// TIA Portal V20 export
FUNCTION_BLOCK "CallUnit"   // FB130, LAD
TITLE = CallUnit
// This block calls all functionality inside the unit.
// stored: IsIECCheckEnabled true, MemoryReserve 100, Namespace Unit1, SetENOAutomatically true
   VAR_INPUT
      safetyReleased : Bool;   // Status from safety program
   END_VAR
   VAR_OUTPUT
      acknowledgeSafety { ExternalWritable := 'False'} : Bool;   // Acknowledge command to the safety program
   END_VAR
   VAR_IN_OUT
      globalStatus : "LAF_typeGeneralStatus";   // Global status
      unitInterface : "LAF_typeUnitInterface";   // Global unit interface
   END_VAR
   VAR
      instManageAlarms { ExternalWritable := 'False'} : "LAF_ManageAlarms";
      instStatusCollector { ExternalWritable := 'False'} : "LUC_StatusCollector";
      instInterfaceManager { ExternalWritable := 'False'} : "LUC_InterfaceManager";
      instUnitModeStateManager { ExternalWritable := 'False'} : "LPMLV2022_UnitModeStateManager";
      instRemoteInterfaceOpcUa { ExternalWritable := 'False'} : "LUC_RemoteCtrl_OpcUa";
      instSignalStack { ExternalWritable := 'False'} : "LUC_SignalStack";
      instUnitModeStateTimes { ExternalWritable := 'False'} : "LPMLV2022_UnitModeStateTimes";
      instUnitModeChangeAllowed { ExternalWritable := 'False'} : "LPMLV2022_UnitModeChangeAllowed";
      instPFEEvents { ExternalWritable := 'False'} : "Unit1.EventsPFE";
      instEQP_Interface_BA030 { ExternalWritable := 'False'} : "LER_EQP_Interface";
      instEQP_Interface_BA040 { ExternalWritable := 'False'} : "LER_EQP_Interface";
      instEQP_Interface_BA100 { S7_SetPoint := 'True'} : "LER_EQP_m_Interface";
      instEQP_Interface_CoveyorA { ExternalWritable := 'False'} : "LER_EQP_Communication";
      instSinaInfeed { ExternalWritable := 'False'} : SinaInfeed;
      statRemoteInterface { ExternalWritable := 'False'} : "LUC_typeCommands";
      statLocalInterface { ExternalWritable := 'False'} : "LUC_typeCommands";
      statEmEnableCheck { ExternalWritable := 'False'} : Array[0..2] of Bool;
      statEmHomeScCheck { ExternalWritable := 'False'} : Array[0..9] of Bool;
      statRunOutStatusCheck { ExternalWritable := 'False'} : Array[0..9] of Bool;
      statEOCStatusCheck { ExternalWritable := 'False'} : Array[0..19] of Bool;
      statPartData { ExternalWritable := 'False'} : Struct
         BA030 : "LER_typePartData";
         BA040 : "LER_typePartData";
      END_STRUCT;
      statDataDelete { ExternalWritable := 'False'} : "LER_typePartData";
      statTonTime { ExternalWritable := 'False'} : Array[0..99] of TON_TIME;
      statTofTime { ExternalWritable := 'False'} : Array[0..9] of TOF_TIME;
      statFlipFlop { ExternalWritable := 'False'} : Array[0..99] of Bool;
      statPulse { ExternalWritable := 'False'} : Array[0..9999] of Bool;
      statNoModeCmd { ExternalWritable := 'False'} : Bool;
      statEnableManualCmds { ExternalWritable := 'False'} : Bool;
      InstLER_FFU_LIU117 { S7_SetPoint := 'True'} : "LER_FFU_LIU117";
      ClearData { S7_SetPoint := 'True'} : "LER_typePartData";
      Data_TrCondition { S7_SetPoint := 'True'} : Array[0..20] of Bool;
      NoData_Alarm : Array[0..20] of Bool;
      statAllEmLinked : Bool;
      citi_Ptrig : Array[0..20] of Bool;
      citiTon : Array[0..20] of TON_TIME;
      citi : Time;
      citiTest : Array[0..20] of Bool;
      instMQTTClient { S7_SetPoint := 'True'} : "LMQTT_Client";
      instPFEUnit { S7_SetPoint := 'True'} : "Unit1.EventsPFE_Unit";
   END_VAR
   VAR_TEMP
      tempUnitFeedback : "LUC_typeEmFeedback";   // Collected commands in the unit, e.g. direct command or commands derived from alarms
      tempProcessCommands : "LUC_typeStateCommands";   // Requested unit state changes by the process
      tempUnitMode : DInt;   // Requested unit mode
      tempUnitModeChangeRequest : Bool;   // Request unit mode
      tempCntrlCmd : DInt;   // Request control command
      tempCmdChangeRequest : Bool;   // Enable change into requested state
      tempSc : Bool;   // State change from FALSE to TRUE (rising edge) triggers state complete signal
      tempEM_Linked_Status_1 : Bool;
      tempEM_Linked_Status_2 : Bool;
      tempDeleteData : Bool;
      tempGather8bits : Array[0..7] of Bool;
   END_VAR
   VAR CONSTANT
      delayTime : Time := T#2s;
      TRUE : Bool := TRUE;
      FALSE : Bool := FALSE;
   END_VAR
   VAR_TEMP   // added for the SCL form of the ladder/FBD networks
      _w1 : Bool;
      _w2 : Bool;
      _w3 : Bool;
      _w4 : Bool;
      _w5 : Bool;
      _w6 : Bool;
      _w7 : Bool;
      _w8 : Bool;
   END_VAR
BEGIN

REGION Network 1: BLOCK INFO HEADER
   // (company) / (C) Copyright (year)
   // ---------------------------------------------------------------------------------
   // Title:                             (Title of this block)
   // Comment/Function: (that is implemented in the block)
   // Library/Family:           (that the source is dedicated to)
   // Author:                        (department / person in charge / contact)
   // Target System:          (test system with FW version)
   // Engineering:              TIA Portal (SW version)
   // Restrictions:               (OB types, etc.)
   // Requirements:           (hardware, technological package, etc.)
   // ---------------------------------------------------------------------------------
   // Change log table:
   // Version          | Date             | Signature      | Expert in charge  | Changes applied ------------------------|----------------------|-------------------------|--------------------------------|-----------------------
   // 001.000.000 | yyyy-mm-dd | 0x00000000 | (name of expert) | First released version
END_REGION

REGION Network 2: DESCRIPTION
   // This is a template block provided by the Automation Framework. It can be used to create an own project.
   // The Block Info Header is prepared to put in your own data.
   // Description of the block could be added here and the docu created by Code2Docu.
END_REGION

REGION Network 3: Simulation
   // If simulation is active on a global level, inherit this status and set simulation active in this unit also. Information is written to DB ControlNodes, from where it is distributed to the equipmemt modules.
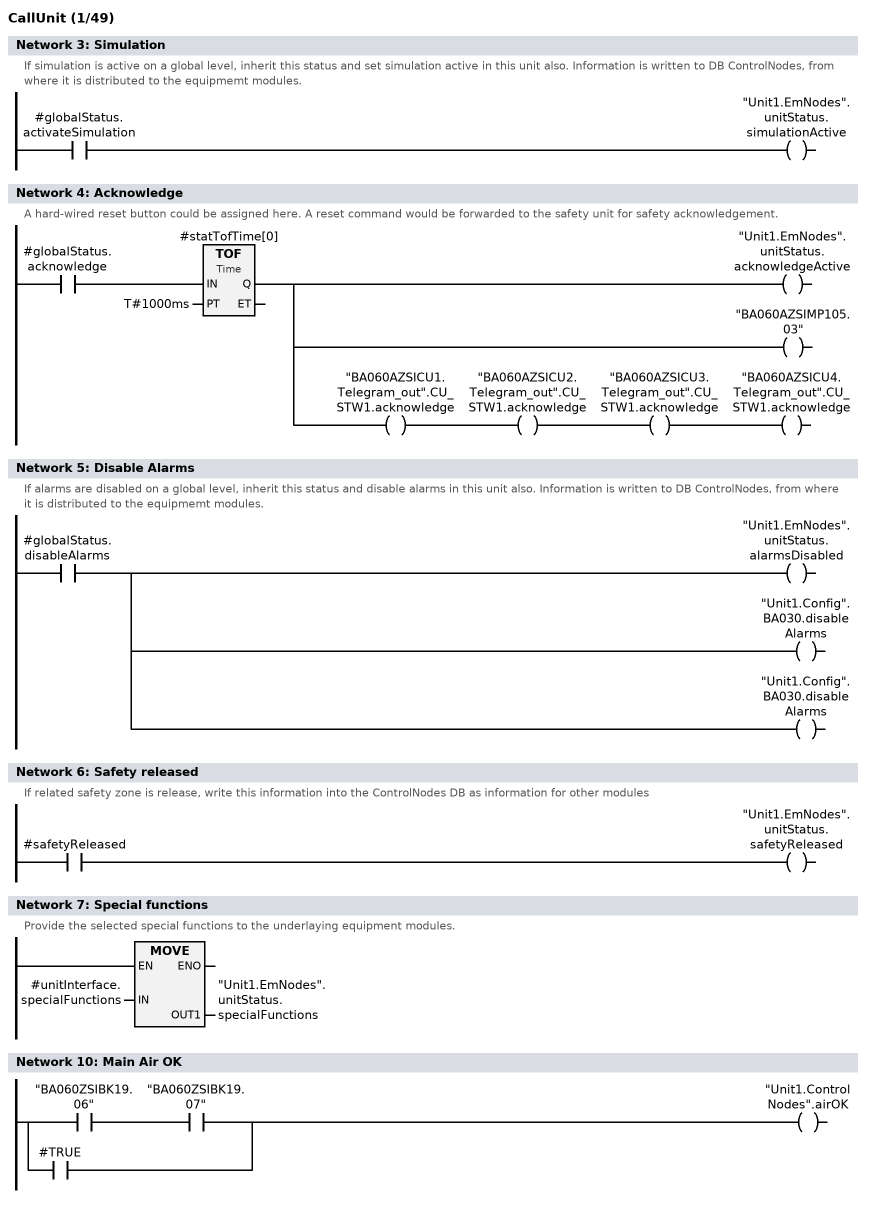
   RUNG wire#powerrail
      Contact( #globalStatus.activateSimulation )
      Coil( "Unit1.EmNodes".unitStatus.simulationActive )
   END_RUNG
   // the same network as SCL:
   "Unit1.EmNodes".unitStatus.simulationActive := #globalStatus.activateSimulation;
END_REGION

REGION Network 4: Acknowledge
   // A hard-wired reset button could be assigned here. A reset command would be forwarded to the safety unit for safety acknowledgement.
   RUNG wire#powerrail
      Contact( #globalStatus.acknowledge )
      { S7_Templates := "time_type := Time" } #statTofTime[0].TOF(pt := T#1000ms, et =>)
      wire#w1
      Coil( "Unit1.EmNodes".unitStatus.acknowledgeActive )
   END_RUNG
   RUNG wire#w1
      Coil( "BA060AZSIMP105.03" )
   END_RUNG
   RUNG wire#w1
      Coil( "BA060AZSICU1.Telegram_out".CU_STW1.acknowledge )
      Coil( "BA060AZSICU2.Telegram_out".CU_STW1.acknowledge )
      Coil( "BA060AZSICU3.Telegram_out".CU_STW1.acknowledge )
      Coil( "BA060AZSICU4.Telegram_out".CU_STW1.acknowledge )
   END_RUNG
   // the same network as SCL:
   #statTofTime[0].TOF(IN := #globalStatus.acknowledge, PT := T#1000ms);
   "Unit1.EmNodes".unitStatus.acknowledgeActive := #statTofTime[0].Q;
   "BA060AZSIMP105.03" := #statTofTime[0].Q;
   "BA060AZSICU1.Telegram_out".CU_STW1.acknowledge := #statTofTime[0].Q;
   "BA060AZSICU2.Telegram_out".CU_STW1.acknowledge := #statTofTime[0].Q;
   "BA060AZSICU3.Telegram_out".CU_STW1.acknowledge := #statTofTime[0].Q;
   "BA060AZSICU4.Telegram_out".CU_STW1.acknowledge := #statTofTime[0].Q;
END_REGION

REGION Network 5: Disable Alarms
   // If alarms are disabled on a global level, inherit this status and disable alarms in this unit also. Information is written to DB ControlNodes, from where it is distributed to the equipmemt modules.
   RUNG wire#powerrail
      Contact( #globalStatus.disableAlarms )
      wire#w1
      Coil( "Unit1.EmNodes".unitStatus.alarmsDisabled )
   END_RUNG
   RUNG wire#w1
      Coil( "Unit1.Config".BA030.disableAlarms )
   END_RUNG
   RUNG wire#w1
      Coil( "Unit1.Config".BA030.disableAlarms )
   END_RUNG
   // the same network as SCL:
   "Unit1.EmNodes".unitStatus.alarmsDisabled := #globalStatus.disableAlarms;
   "Unit1.Config".BA030.disableAlarms := #globalStatus.disableAlarms;
   "Unit1.Config".BA030.disableAlarms := #globalStatus.disableAlarms;
END_REGION

REGION Network 6: Safety released
   // If related safety zone is release, write this information into the ControlNodes DB as information for other modules
   RUNG wire#powerrail
      Contact( #safetyReleased )
      Coil( "Unit1.EmNodes".unitStatus.safetyReleased )
   END_RUNG
   // the same network as SCL:
   "Unit1.EmNodes".unitStatus.safetyReleased := #safetyReleased;
END_REGION

REGION Network 7: Special functions
   // Provide the selected special functions to the underlaying equipment modules.
   RUNG wire#powerrail
      Move(in := #unitInterface.specialFunctions, out1 => "Unit1.EmNodes".unitStatus.specialFunctions)
   END_RUNG
   // the same network as SCL:
   "Unit1.EmNodes".unitStatus.specialFunctions := #unitInterface.specialFunctions;
END_REGION

REGION Network 8 (SCL): Electric Power CB
   "Unit1.ControlNodes".fuse[0] := "BA060AZSIMP101.00"; //KISTLER 100KN PRESS POWER TRIPPED E202CB
   "Unit1.ControlNodes".fuse[1] := "BA060AZSIMP101.01"; //KISTLER 100KN PRESS POWER TRIPPED E208CB
   "Unit1.ControlNodes".fuse[2] := "BA060AZSIMP101.02"; //KISTLER 30KN PRESS POWER TRIPPED E214CB
   "Unit1.ControlNodes".fuse[3] := "BA060AZSIMP101.03"; //SPARE
   "Unit1.ControlNodes".fuse[4] := "BA060AZSIMP101.04"; //SPARE
   "Unit1.ControlNodes".fuse[5] := "BA060AZSIMP101.05"; //E8404PWS CONTROLLER POWER SMPS AC POWER TRIPPED E320CB
   "Unit1.ControlNodes".fuse[6] := "BA060AZSIMP101.06"; //E8704PWS SAFETY POWER SMPS AC POWER TRIPPED E326CB
   "Unit1.ControlNodes".fuse[7] := "BA060AZSIMP101.07"; //E8804PWS CONTRL POWER SMPS AC POWER TRIPPED E332CB
   "Unit1.ControlNodes".fuse[8] := "BA060AZSIMP101.10"; //PROCESSOR POWER ON TIPPRED E4120CB
   "Unit1.ControlNodes".fuse[9] := "BA060AZSIMP101.11"; //PROGRAMING POWER OUTLET TRPPED E4126CB
   "Unit1.ControlNodes".fuse[10] := "BA060AZSIMP101.12"; //SPARE
   "Unit1.ControlNodes".fuse[11] := "BA060AZSIMP101.13"; //PANEL LED POWER TRIPPED E4304CB
   "Unit1.ControlNodes".fuse[12] := "BA060AZSIMP101.14"; //SPARE
   "Unit1.ControlNodes".fuse[13] := "BA060AZSIMP101.16"; //CONTROL LEVEL HUB POWER TRIPPED E4420CB
   "Unit1.ControlNodes".fuse[14] := "BA060AZSIMP101.17"; //MAIN HMI POWER TRIPPED E4426CB
   "Unit1.ControlNodes".fuse[15] := "BA060AZSIMP101.20"; //PORTABLE HMI POWER TIPPED E4432CB
   "Unit1.ControlNodes".fuse[16] := "BA060AZSIMP101.21"; //PORTABLE HMI POWER TIPPED E4456CB
   "Unit1.ControlNodes".fuse[17] := "BA060AZSIMP101.22"; //120VAC HEATER-1 POWER TR PRIMARY TRIPPED E5100CB
   "Unit1.ControlNodes".fuse[18] := "BA060AZSIMP101.23"; //SPARE
   "Unit1.ControlNodes".fuse[19] := "BA060AZSIMP101.24"; //SPARE
   "Unit1.ControlNodes".fuse[20] := "BA060AZSIMP101.25"; //UPPER 1-1 HEATER POWER TRIPPED E5156CB
   "Unit1.ControlNodes".fuse[21] := "BA060AZSIMP101.26"; //UPPER 1-2 HEATER POWER TRIPPED E5162CB
   "Unit1.ControlNodes".fuse[22] := "BA060AZSIMP101.27"; //LOWER 1-1 HEATER POWER TRIPPED E5168CB
   "Unit1.ControlNodes".fuse[23] := "BA060AZSIMP101.30"; //LOWER 1-2 HEATER POWER TRIPPED E5174CB
   "Unit1.ControlNodes".fuse[24] := "BA060AZSIMP101.31"; //LOWER 1-3 HEATER POWER TRIPPED E5180CB
   "Unit1.ControlNodes".fuse[25] := "BA060AZSIMP101.32"; //SPARE
   "Unit1.ControlNodes".fuse[26] := "BA060AZSIMP101.33"; //120VAC HEATER-2 POWER TR PRIMARY TRIPPED E6100CB
   "Unit1.ControlNodes".fuse[27] := "BA060AZSIMP101.34"; //SPARE
   "Unit1.ControlNodes".fuse[28] := "BA060AZSIMP101.35"; //SPARE
   "Unit1.ControlNodes".fuse[29] := "BA060AZSIMP101.36"; //UPPER 2-1 HEATER POWER TRIPPED E6156CB
   "Unit1.ControlNodes".fuse[30] := "BA060AZSIMP101.37"; //UPPER 2-2 HEATER POWER TRIPPED E6162CB
   "Unit1.ControlNodes".fuse[31] := "BA060AZSIMP102.00"; //LOWER 2-1 HEATER POWER TRIPPED E6168CB
   "Unit1.ControlNodes".fuse[32] := "BA060AZSIMP102.01"; //LOWER 2-2 HEATER POWER TRIPPED E6174CB
   "Unit1.ControlNodes".fuse[33] := "BA060AZSIMP102.02"; //LOWER 2-3 HEATER POWER TRIPPED E6180CB
   "Unit1.ControlNodes".fuse[34] := "BA060AZSIMP102.03"; //SPARE
   "Unit1.ControlNodes".fuse[35] := "BA060AZSIMP102.04"; //120VAC CONTROL POWER TR PRIMARY TRIPPED E7100CB
   "Unit1.ControlNodes".fuse[36] := "BA060AZSIMP102.05"; //120VAC CONTROL POWER TR SECONDARY TRIPPED E7110CB
   "Unit1.ControlNodes".fuse[37] := "BA060AZSIMP102.06"; //CONTROL POWER ON TRIPPED E7116CB
   "Unit1.ControlNodes".fuse[38] := "BA060AZSIMP102.07"; //MOTOR PANEL CONTROL POWER TRIPPED E7154CB
   "Unit1.ControlNodes".fuse[39] := "BA060AZSIMP102.10"; //POWER STRIP OUTLET POWER TRIPPED E7160CB
   "Unit1.ControlNodes".fuse[40] := "BA060AZSIMP102.11"; //POWER STRIP OUTLET POWER TRIPPED E7166CB
   "Unit1.ControlNodes".fuse[41] := "BA060AZSIMP102.12"; //QR LASER MARKING TRIPPED E7172CB
   "Unit1.ControlNodes".fuse[42] := "BA060AZSIMP102.13"; //HI-POT TESTER POWER TRIPPED E7178CB
   "Unit1.ControlNodes".fuse[43] := "BA060AZSIMP102.14"; //FFU-1 POWER TRIPPED E7222CB
   "Unit1.ControlNodes".fuse[44] := "BA060AZSIMP102.15"; //UPPER 1-1 TEMPERATURE CONTROLLER POWER TRIPPED E5206CB
   "Unit1.ControlNodes".fuse[45] := "BA060AZSIMP102.16"; //UPPER 1-2 TEMPERATURE CONTROLLER POWER TRIPPED E5212CB
   "Unit1.ControlNodes".fuse[46] := "BA060AZSIMP102.17"; //LOWER 1-1 TEMPERATURE CONTROLLER POWER TRIPPED E5218CB
   "Unit1.ControlNodes".fuse[47] := "BA060AZSIMP102.20"; //LOWER 1-2 TEMPERATURE CONTROLLER POWER TRIPPED E5224CB
   "Unit1.ControlNodes".fuse[48] := "BA060AZSIMP102.21"; //LOWER 1-3 TEMPERATURE CONTROLLER POWER TRIPPED E5230CB
   "Unit1.ControlNodes".fuse[49] := "BA060AZSIMP102.22"; //UPPER 2-1 TEMPERATURE CONTROLLER POWER TRIPPED E6206CB
   "Unit1.ControlNodes".fuse[50] := "BA060AZSIMP102.23"; //UPPER 2-2 TEMPERATURE CONTROLLER POWER TRIPPED E6212CB
   "Unit1.ControlNodes".fuse[51] := "BA060AZSIMP102.24"; //LOWER 2-1 TEMPERATURE CONTROLLER POWER TRIPPED E6218CB
   "Unit1.ControlNodes".fuse[52] := "BA060AZSIMP102.25"; //LOWER 2-2 TEMPERATURE CONTROLLER POWER TRIPPED E6224CB
   "Unit1.ControlNodes".fuse[53] := "BA060AZSIMP102.26"; //LOWER 2-3 TEMPERATURE CONTROLLER POWER TRIPPED E6230CB
   "Unit1.ControlNodes".fuse[54] := "BA060AZSIMP102.27"; //SPARE
   "Unit1.ControlNodes".fuse[55] := "BA060AZSIMP102.31"; //ET200MP I/O OUTPUT POWER TRIPPED E8154CB
   "Unit1.ControlNodes".fuse[56] := "BA060AZSIMP102.32"; //JUNCTION BOX CONTROL POWER TRIPPED E8180CB
   "Unit1.ControlNodes".fuse[57] := "BA060AZSIMP102.33"; //CLASS 2 SMPS POWER TRIPPED E8204CB
   "Unit1.ControlNodes".fuse[58] := "BA060AZSIMP102.35"; //ET200ECO PN-1 POWER TRIPPED E8220CB
   "Unit1.ControlNodes".fuse[59] := "BA060AZSIMP102.36"; //ET200ECO PN-2 POWER TRIPPED E8224CB
   "Unit1.ControlNodes".fuse[60] := "BA060AZSIMP102.37"; //ET200ECO PN-3 POWER TRIPPED E8228CB
   "Unit1.ControlNodes".fuse[61] := "BA060AZSIMP103.00"; //ET200ECO PN-4 POWER TRIPPED E8232CB
   "Unit1.ControlNodes".fuse[62] := "BA060AZSIMP103.01"; //PANEL FAN POWER TRIPPED E8304CB
   "Unit1.ControlNodes".fuse[63] := "BA060AZSIMP103.02"; //SPARE
   "Unit1.ControlNodes".fuse[64] := "BA060AZSIMP103.04"; //CONTROLLER DC POWER TRIPPED E8406CB
   "Unit1.ControlNodes".fuse[65] := "BA060AZSIMP103.05"; //KISTLER CONTROL POWER TRIPPED E8416CB
   "Unit1.ControlNodes".fuse[66] := "BA060AZSIMP103.06"; //MANIFOLD-1 POWER TRIPPED E8422CB
   "Unit1.ControlNodes".fuse[67] := "BA060AZSIMP103.07"; //MANIFOLD-2 POWER TRIPPED E8430CB
   "Unit1.ControlNodes".fuse[68] := "BA060AZSIMP103.10"; //QR READER POWER TRIPPED E8456CB
   "Unit1.ControlNodes".fuse[69] := "BA060AZSIMP103.11"; //QR READER POWER TRIPPED E8462CB
   "Unit1.ControlNodes".fuse[70] := "BA060AZSIMP103.12"; //HANDY QR READER POWER TRIPPED E8468CB
   "Unit1.ControlNodes".fuse[71] := "BA060AZSIMP103.13"; //PROFINET CONVERTER POWER TRIPPED E8474CB
   "Unit1.ControlNodes".fuse[72] := "BA060AZSIMP103.14"; //MONITORING RELAY POWER TRIPPED E8504CB
   "Unit1.ControlNodes".fuse[73] := "BA060AZSIMP103.15"; //SPARE
   "Unit1.ControlNodes".fuse[74] := "BA060AZSIMP103.17"; //SAFETY DC POWER TRIPPED E8706CB
   "Unit1.ControlNodes".fuse[75] := "BA060AZSIMP103.20"; //ET200SP I/O SAFETY POWER TRIPPED E8716CB
   "Unit1.ControlNodes".fuse[76] := "BA060AZSIMP103.21"; //JUNCTION BOX CONTROL POWER TRIPPED E8736CB
   "Unit1.ControlNodes".fuse[77] := "BA060AZSIMP103.22"; //ET200ECO PN SAFETYT-1 POWER TRIPPED E8756CB
   "Unit1.ControlNodes".fuse[78] := "BA060AZSIMP103.23"; //ET200ECO PN SAFETYT-2 POWER TRIPPED E8762CB
   "Unit1.ControlNodes".fuse[79] := "BA060AZSIMP103.24"; //SPARE
   "Unit1.ControlNodes".fuse[80] := "BA060AZSIMP103.26"; //CONTROL DC POWER TRIPPED E8806CB
   "Unit1.ControlNodes".fuse[81] := "BA060AZSIMP103.27"; //JUNCTION BOX CONTROL POWER TRIPPED E8816CB
   "Unit1.ControlNodes".fuse[82] := "BA060AZSIMP103.30"; //DRIVE-CLIQ HUB POWER TRIPPED E8822CB
   "Unit1.ControlNodes".fuse[83] := "BA060AZSIMP103.31"; //EQUIPMENT LED POWER TRIPPED E8828CB
   "Unit1.ControlNodes".fuse[84] := "BA060AZSISP501.00"; //SPARE
   "Unit1.ControlNodes".fuse[85] := "BA060AZSISP501.01"; //SAFETY DC POWER TRIPPED E218CB
   "Unit1.ControlNodes".fuse[86] := "BA060AZSISP501.02"; //CLASS 2 SMPS POWER TRIPPED E308CB
   "Unit1.ControlNodes".fuse[87] := "BA060AZSISP501.04"; //ET200ECO PN-1 POWER TRIPPED E324CB
   "Unit1.ControlNodes".fuse[88] := "BA060AZSISP501.05"; //ET200ECO PN-2 POWER TRIPPED E328CB
   "Unit1.ControlNodes".fuse[89] := "BA060AZSISP501.06"; //ET200ECO PN-3 POWER TRIPPED E332CB
   "Unit1.ControlNodes".fuse[90] := "BA060AZSISP501.07"; //ET200ECO PN-4 POWER TRIPPED E336CB
   "Unit1.ControlNodes".fuse[91] := "BA060AZSICU1.Telegram_In".E_DIGITAL.digitalInput0; //MOTOR POWER MC FEEDBACK
   "Unit1.ControlNodes".fuse[92] := "BA060AZSICU1.Telegram_In".E_DIGITAL.digitalInput1; //MOTOR POWER TRIPPED E202CB
   "Unit1.ControlNodes".fuse[93] := "BA060AZSICU1.Telegram_In".E_DIGITAL.digitalInput2; //MAIN CONTROL PANEL MAIN POWER TRIPPED E208CB
   "Unit1.ControlNodes".fuse[94] := "BA060AZSICU1.Telegram_In".E_DIGITAL.digitalInput3; //E6104PWS CONTROL POWER SMPS AC POWER TRIPPED E314CB
   "Unit1.ControlNodes".fuse[95] := "BA060AZSICU1.Telegram_In".E_DIGITAL.digitalInput4; //JROUT P&P Y-AXIS POWER TR PRIMARY TRIPPED E400CB
   "Unit1.ControlNodes".fuse[96] := "BA060AZSICU1.Telegram_In".E_DIGITAL.digitalInput5; //JROUT P&P Y-AXIS POWER TR ECONDARY TRIPPED E410CB
   "Unit1.ControlNodes".fuse[97] := "BA060AZSICU1.Telegram_In".E_DIGITAL.digitalInput6; //INS PROCESS P&P X-AXIS POWER TR PRIMARY TRIPPED E500CB
   "Unit1.ControlNodes".fuse[98] := "BA060AZSICU1.Telegram_In".E_DIGITAL.digitalInput7; //INS PROCESS P&P X-AXIS POWER TR ECONDARY TRIPPED E510CB
   "Unit1.ControlNodes".fuse[99] := "BA060AZSICU2.Telegram_In".E_DIGITAL.digitalInput0; //JR UNLOADING Y-AXIS POWER TR PRIMARY TRIPPED E600CB
   "Unit1.ControlNodes".fuse[100] := "BA060AZSICU2.Telegram_In".E_DIGITAL.digitalInput1; //JR UNLOADING Y-AXIS POWER TR ECONDARY TRIPPED E610CB
   "Unit1.ControlNodes".fuse[101] := "BA060AZSICU2.Telegram_In".E_DIGITAL.digitalInput2; //POWER METER POWER TRIIPED E720CB
   "Unit1.ControlNodes".fuse[102] := "BA060AZSICU2.Telegram_In".E_DIGITAL.digitalInput3; //POWER METER CONTROL POWER TRIIPED E726CB
   "Unit1.ControlNodes".fuse[103] := "BA060AZSICU2.Telegram_In".E_DIGITAL.digitalInput4; //JR OUT P&P 1 Y-AXIS POWER ON TRIPPED E2004CB
   "Unit1.ControlNodes".fuse[104] := "BA060AZSICU2.Telegram_In".E_DIGITAL.digitalInput5; //JR OUT P&P 2 Y-AXIS POWER ON TRIPPED E2104CB
   "Unit1.ControlNodes".fuse[105] := "BA060AZSICU2.Telegram_In".E_DIGITAL.digitalInput6; //INS PROCESS P&P 1 X-AXIS POWER ON TRIPPED E2204CB
   "Unit1.ControlNodes".fuse[106] := "BA060AZSICU2.Telegram_In".E_DIGITAL.digitalInput7; //INS PROCESS P&P 2 X-AXIS POWER ON TRIPPED E2304CB
   "Unit1.ControlNodes".fuse[107] := "BA060AZSICU3.Telegram_In".E_DIGITAL.digitalInput0; //JR UNLOADING Y-AXIS POWER ON TRIPPED E2404CB
   "Unit1.ControlNodes".fuse[108] := "BA060AZSICU3.Telegram_In".E_DIGITAL.digitalInput1; //MOTOR POWER MC COIL POWER TRIPPED E6156CB
   "Unit1.ControlNodes".fuse[109] := "BA060AZSICU3.Telegram_In".E_DIGITAL.digitalInput2; //PROCESSOR POWER ON TRIPPRED E4116CB
   "Unit1.ControlNodes".fuse[110] := "BA060AZSICU3.Telegram_In".E_DIGITAL.digitalInput3; //MAIN CONTROL PANEL HOT POWER TRIPPED E4156CB
   "Unit1.ControlNodes".fuse[111] := "BA060AZSICU3.Telegram_In".E_DIGITAL.digitalInput4; //SYSTEM LEVEL HUB POWER TRIPPED E4162CB
   "Unit1.ControlNodes".fuse[112] := "BA060AZSICU3.Telegram_In".E_DIGITAL.digitalInput5; //PANEL LED POWER TRIPPED E4304CB
   "Unit1.ControlNodes".fuse[113] := "BA060AZSICU3.Telegram_In".E_DIGITAL.digitalInput6; //CONTROL POWER TRIPPED E5110CB
   "Unit1.ControlNodes".fuse[114] := "BA060AZSICU3.Telegram_In".E_DIGITAL.digitalInput7; //CONTROL POWER ON TRIPPED E5120CB
   "Unit1.ControlNodes".fuse[115] := "BA060AZSICU4.Telegram_In".E_DIGITAL.digitalInput1; //SERVON CONTROL POWER TRIPPED E6122CB
   "Unit1.ControlNodes".fuse[116] := "BA060AZSICU4.Telegram_In".E_DIGITAL.digitalInput2; //SERVO CONTROL UNIT CONTROL POWER TRIPPED E6128CB
   "Unit1.ControlNodes".fuse[117] := "BA060AZSICU4.Telegram_In".E_DIGITAL.digitalInput3; //PANEL FAN POWER TRIPPED E6204CB
   "Unit1.ControlNodes".fuse[118] := "BA060AZSICU4.Telegram_In".E_DIGITAL.digitalInput4; //SPARE
   "Unit1.ControlNodes".fuse[119] := "BA060AZSICU4.Telegram_In".E_DIGITAL.digitalInput5; //SPARE
   "Unit1.ControlNodes".fuse[120] := "BA060AZSICU4.Telegram_In".E_DIGITAL.digitalInput6; //SPARE
   "Unit1.ControlNodes".fuse[121] := "BA060AZSICU4.Telegram_In".E_DIGITAL.digitalInput7; //SPARE
END_REGION

REGION Network 9 (SCL): Electric Power PWS
   "Unit1.ControlNodes".pws[0] := "BA060AZSIMP101.15"; //PLC POWER SMPS DC OK E4404PWS
   "Unit1.ControlNodes".pws[1] := "BA060AZSIMP102.30"; //CONTROL POWER SMPS DC OK E8104PWS
   "Unit1.ControlNodes".pws[2] := "BA060AZSIMP102.34"; //CLASS 2 SMPS MONITORING E8206PWS
   "Unit1.ControlNodes".pws[3] := "BA060AZSIMP103.03"; //CONTROLLER POWER SMPS DC OK E8404PWS
   "Unit1.ControlNodes".pws[4] := "BA060AZSIMP103.16"; //SAFETY POWER SMPS DC OK E8704PWS
   "Unit1.ControlNodes".pws[5] := "BA060AZSIMP103.25"; //COONTRL POWER SMPS DC OK E8804PWS
   "Unit1.ControlNodes".pws[6] := "BA060AZSISP501.03"; //CLASS 2 SMPS MONITORING E310PWS
   "Unit1.ControlNodes".pws[7] := "BA060AZSICU4.Telegram_In".E_DIGITAL.digitalInput0; //CONTROL POWER SMPS DC OK E6104PWS
END_REGION

REGION Network 10: Main Air OK
   RUNG wire#powerrail
      Contact( "BA060ZSIBK19.06" )
      Contact( "BA060ZSIBK19.07" )
      wire#w1
      Coil( "Unit1.ControlNodes".airOK )
   END_RUNG
   RUNG wire#powerrail
      Contact( #TRUE )
   END_RUNG wire#w1
   // the same network as SCL:
   "Unit1.ControlNodes".airOK := ("BA060ZSIBK19.06" AND "BA060ZSIBK19.07") OR #TRUE;
END_REGION

REGION Network 11: Collect Alarms
   // Add events here that trigger alarms and lead to the respective commands to the unit. It is possible to trigger alarms, set unit commands or do both for the specific event
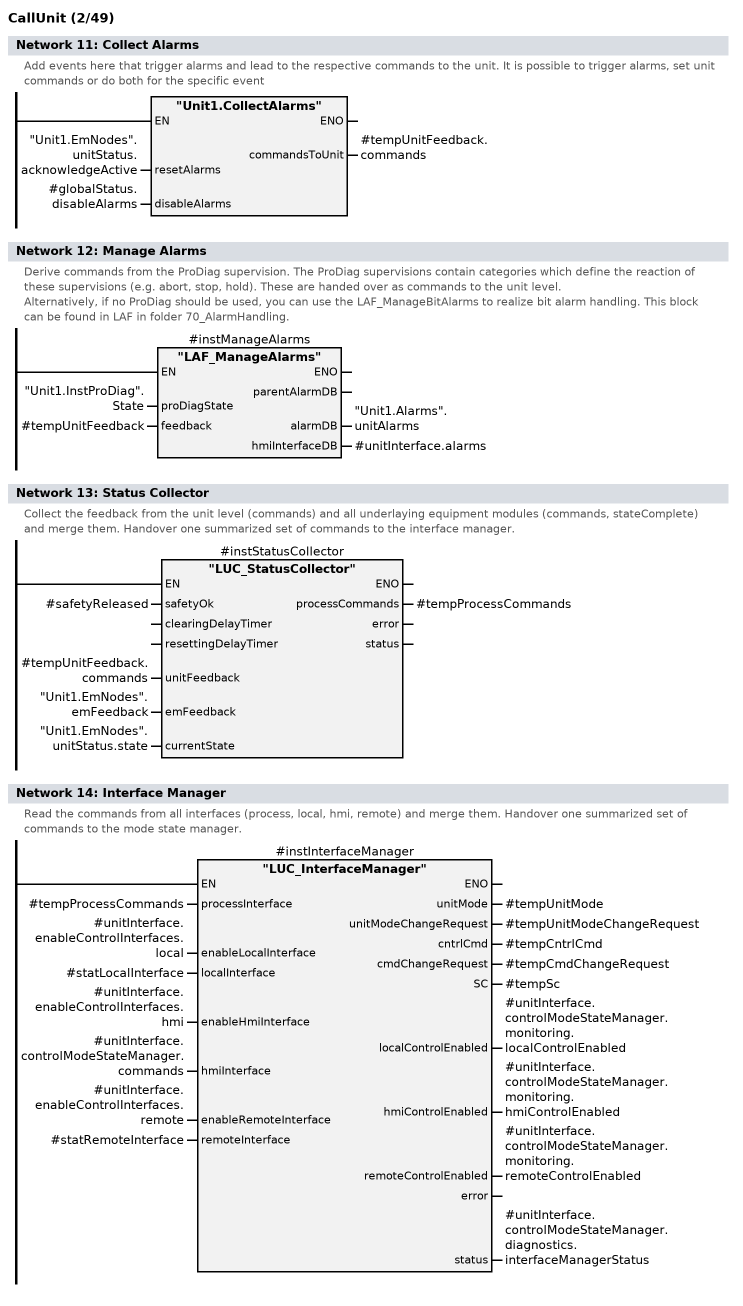
   RUNG wire#powerrail
      "Unit1.CollectAlarms"(resetAlarms := "Unit1.EmNodes".unitStatus.acknowledgeActive, disableAlarms := #globalStatus.disableAlarms, commandsToUnit => #tempUnitFeedback.commands)
   END_RUNG
   // the same network as SCL:
   "Unit1.CollectAlarms"(resetAlarms := "Unit1.EmNodes".unitStatus.acknowledgeActive,
                         disableAlarms := #globalStatus.disableAlarms,
                         commandsToUnit => #tempUnitFeedback.commands);
END_REGION

REGION Network 12: Manage Alarms
   // Derive commands from the ProDiag supervision. The ProDiag supervisions contain categories which define the reaction of these supervisions (e.g. abort, stop, hold). These are handed over as commands to the unit level.
   // Alternatively, if no ProDiag should be used, you can use the LAF_ManageBitAlarms to realize bit alarm handling. This block can be found in LAF in folder 70_AlarmHandling.
   RUNG wire#powerrail
      #instManageAlarms(proDiagState := "Unit1.InstProDiag".State, feedback := #tempUnitFeedback, parentAlarmDB =>, alarmDB => "Unit1.Alarms".unitAlarms, hmiInterfaceDB => #unitInterface.alarms)
   END_RUNG
   // the same network as SCL:
   #instManageAlarms(proDiagState := "Unit1.InstProDiag".State,   // "LAF_ManageAlarms"
                     feedback := #tempUnitFeedback,
                     alarmDB => "Unit1.Alarms".unitAlarms,
                     hmiInterfaceDB => #unitInterface.alarms);
END_REGION

REGION Network 13: Status Collector
   // Collect the feedback from the unit level (commands) and all underlaying equipment modules (commands, stateComplete) and merge them. Handover one summarized set of commands to the interface manager.
   RUNG wire#powerrail
      #instStatusCollector(safetyOk := #safetyReleased, clearingDelayTimer :=, resettingDelayTimer :=, unitFeedback := #tempUnitFeedback.commands, emFeedback := "Unit1.EmNodes".emFeedback, currentState := "Unit1.EmNodes".unitStatus.state, processCommands => #tempProcessCommands, error =>, status =>)
   END_RUNG
   // the same network as SCL:
   #instStatusCollector(safetyOk := #safetyReleased,   // "LUC_StatusCollector"
                        unitFeedback := #tempUnitFeedback.commands,
                        emFeedback := "Unit1.EmNodes".emFeedback,
                        currentState := "Unit1.EmNodes".unitStatus.state,
                        processCommands => #tempProcessCommands);
END_REGION

REGION Network 14: Interface Manager
   // Read the commands from all interfaces (process, local, hmi, remote) and merge them. Handover one summarized set of commands to the mode state manager.
   RUNG wire#powerrail
      #instInterfaceManager(processInterface := #tempProcessCommands, enableLocalInterface := #unitInterface.enableControlInterfaces.local, localInterface := #statLocalInterface, enableHmiInterface := #unitInterface.enableControlInterfaces.hmi, hmiInterface := #unitInterface.controlModeStateManager.commands, enableRemoteInterface := #unitInterface.enableControlInterfaces.remote, remoteInterface := #statRemoteInterface, unitMode => #tempUnitMode, unitModeChangeRequest => #tempUnitModeChangeRequest, cntrlCmd => #tempCntrlCmd, cmdChangeRequest => #tempCmdChangeRequest, SC => #tempSc, localControlEnabled => #unitInterface.controlModeStateManager.monitoring.localControlEnabled, hmiControlEnabled => #unitInterface.controlModeStateManager.monitoring.hmiControlEnabled, remoteControlEnabled => #unitInterface.controlModeStateManager.monitoring.remoteControlEnabled, error =>, status => #unitInterface.controlModeStateManager.diagnostics.interfaceManagerStatus)
   END_RUNG
   // the same network as SCL:
   #instInterfaceManager(processInterface := #tempProcessCommands,   // "LUC_InterfaceManager"
                         enableLocalInterface := #unitInterface.enableControlInterfaces.local,
                         localInterface := #statLocalInterface,
                         enableHmiInterface := #unitInterface.enableControlInterfaces.hmi,
                         hmiInterface := #unitInterface.controlModeStateManager.commands,
                         enableRemoteInterface := #unitInterface.enableControlInterfaces.remote,
                         remoteInterface := #statRemoteInterface,
                         unitMode => #tempUnitMode,
                         unitModeChangeRequest => #tempUnitModeChangeRequest,
                         cntrlCmd => #tempCntrlCmd,
                         cmdChangeRequest => #tempCmdChangeRequest,
                         SC => #tempSc,
                         localControlEnabled => #unitInterface.controlModeStateManager.monitoring.localControlEnabled,
                         hmiControlEnabled => #unitInterface.controlModeStateManager.monitoring.hmiControlEnabled,
                         remoteControlEnabled => #unitInterface.controlModeStateManager.monitoring.remoteControlEnabled,
                         status => #unitInterface.controlModeStateManager.diagnostics.interfaceManagerStatus);
END_REGION

REGION Network 15: Mode and State Manager
   // Determine unit mode and state based on the collected commands and status
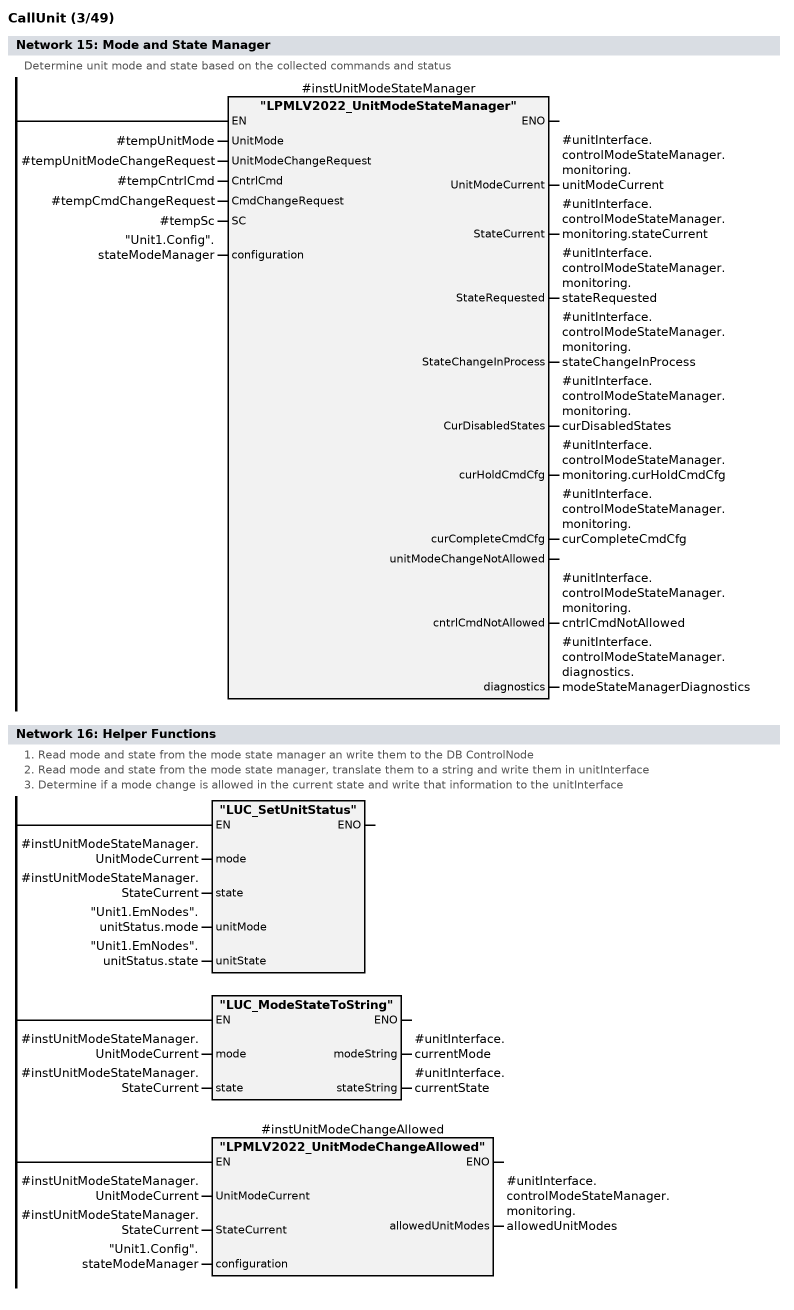
   RUNG wire#powerrail
      #instUnitModeStateManager(UnitMode := #tempUnitMode, UnitModeChangeRequest := #tempUnitModeChangeRequest, CntrlCmd := #tempCntrlCmd, CmdChangeRequest := #tempCmdChangeRequest, SC := #tempSc, configuration := "Unit1.Config".stateModeManager, UnitModeCurrent => #unitInterface.controlModeStateManager.monitoring.unitModeCurrent, StateCurrent => #unitInterface.controlModeStateManager.monitoring.stateCurrent, StateRequested => #unitInterface.controlModeStateManager.monitoring.stateRequested, StateChangeInProcess => #unitInterface.controlModeStateManager.monitoring.stateChangeInProcess, CurDisabledStates => #unitInterface.controlModeStateManager.monitoring.curDisabledStates, curHoldCmdCfg => #unitInterface.controlModeStateManager.monitoring.curHoldCmdCfg, curCompleteCmdCfg => #unitInterface.controlModeStateManager.monitoring.curCompleteCmdCfg, unitModeChangeNotAllowed =>, cntrlCmdNotAllowed => #unitInterface.controlModeStateManager.monitoring.cntrlCmdNotAllowed, diagnostics => #unitInterface.controlModeStateManager.diagnostics.modeStateManagerDiagnostics)
   END_RUNG
   // the same network as SCL:
   #instUnitModeStateManager(UnitMode := #tempUnitMode,   // "LPMLV2022_UnitModeStateManager"
                           UnitModeChangeRequest := #tempUnitModeChangeRequest,
                           CntrlCmd := #tempCntrlCmd,
                           CmdChangeRequest := #tempCmdChangeRequest,
                           SC := #tempSc,
                           configuration := "Unit1.Config".stateModeManager,
                           UnitModeCurrent => #unitInterface.controlModeStateManager.monitoring.unitModeCurrent,
                           StateCurrent => #unitInterface.controlModeStateManager.monitoring.stateCurrent,
                           StateRequested => #unitInterface.controlModeStateManager.monitoring.stateRequested,
                           StateChangeInProcess => #unitInterface.controlModeStateManager.monitoring.stateChangeInProcess,
                           CurDisabledStates => #unitInterface.controlModeStateManager.monitoring.curDisabledStates,
                           curHoldCmdCfg => #unitInterface.controlModeStateManager.monitoring.curHoldCmdCfg,
                           curCompleteCmdCfg => #unitInterface.controlModeStateManager.monitoring.curCompleteCmdCfg,
                           cntrlCmdNotAllowed => #unitInterface.controlModeStateManager.monitoring.cntrlCmdNotAllowed,
                           diagnostics => #unitInterface.controlModeStateManager.diagnostics.modeStateManagerDiagnostics);
END_REGION

REGION Network 16: Helper Functions
   // 1. Read mode and state from the mode state manager an write them to the DB ControlNode
   // 2. Read mode and state from the mode state manager, translate them to a string and write them in unitInterface
   // 3. Determine if a mode change is allowed in the current state and write that information to the unitInterface
   RUNG wire#powerrail
      "LUC_SetUnitStatus"(mode := #instUnitModeStateManager.UnitModeCurrent, state := #instUnitModeStateManager.StateCurrent, unitMode := "Unit1.EmNodes".unitStatus.mode, unitState := "Unit1.EmNodes".unitStatus.state)
   END_RUNG
   RUNG wire#powerrail
      "LUC_ModeStateToString"(mode := #instUnitModeStateManager.UnitModeCurrent, state := #instUnitModeStateManager.StateCurrent, modeString => #unitInterface.currentMode, stateString => #unitInterface.currentState)
   END_RUNG
   RUNG wire#powerrail
      #instUnitModeChangeAllowed(UnitModeCurrent := #instUnitModeStateManager.UnitModeCurrent, StateCurrent := #instUnitModeStateManager.StateCurrent, configuration := "Unit1.Config".stateModeManager, allowedUnitModes => #unitInterface.controlModeStateManager.monitoring.allowedUnitModes)
   END_RUNG
   // the same network as SCL:
   "LUC_SetUnitStatus"(mode := #instUnitModeStateManager.UnitModeCurrent,
                       state := #instUnitModeStateManager.StateCurrent,
                       unitMode := "Unit1.EmNodes".unitStatus.mode,
                       unitState := "Unit1.EmNodes".unitStatus.state);
   "LUC_ModeStateToString"(mode := #instUnitModeStateManager.UnitModeCurrent,
                           state := #instUnitModeStateManager.StateCurrent,
                           modeString => #unitInterface.currentMode,
                           stateString => #unitInterface.currentState);
   #instUnitModeChangeAllowed(UnitModeCurrent := #instUnitModeStateManager.UnitModeCurrent,   // "LPMLV2022_UnitModeChangeAllowed"
                           StateCurrent := #instUnitModeStateManager.StateCurrent,
                           configuration := "Unit1.Config".stateModeManager,
                           allowedUnitModes => #unitInterface.controlModeStateManager.monitoring.allowedUnitModes);
END_REGION

REGION Network 17: History
   // Update the mode and state history. When mode or state change occur, save current mode and state in history[0] and the previous ones in ascending order.
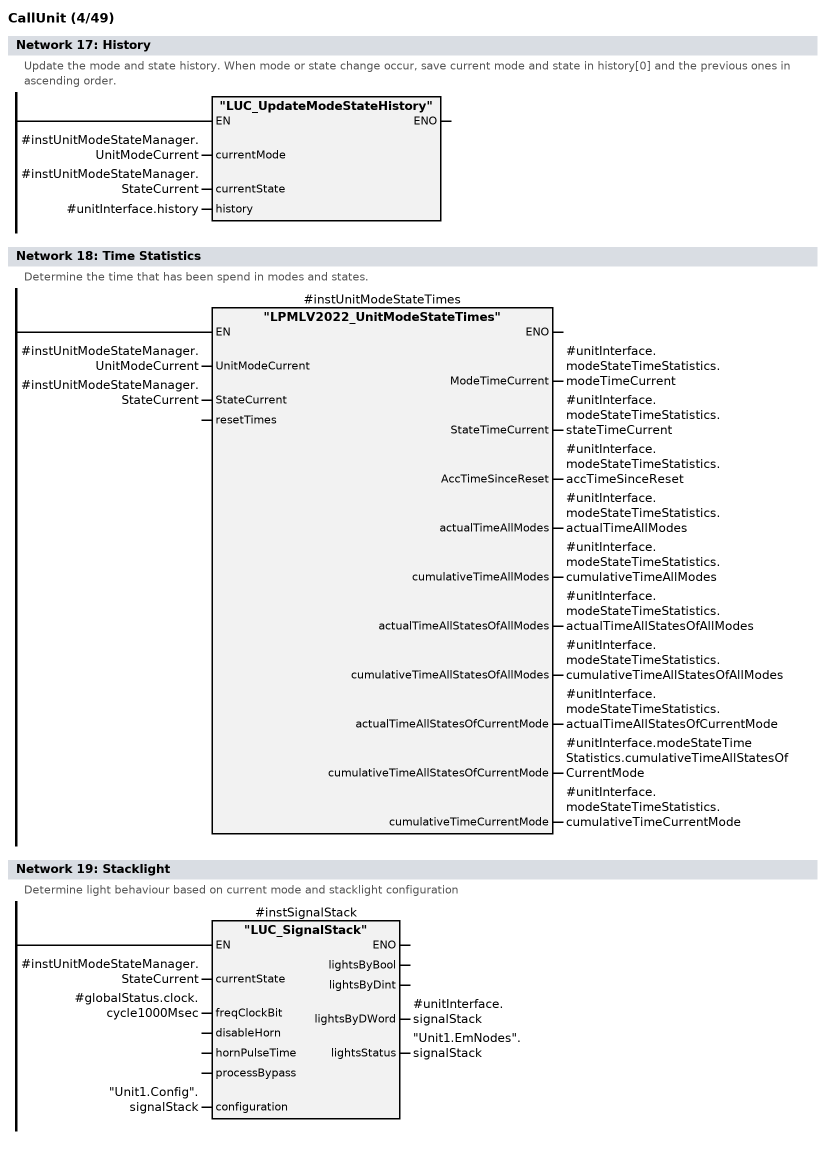
   RUNG wire#powerrail
      "LUC_UpdateModeStateHistory"(currentMode := #instUnitModeStateManager.UnitModeCurrent, currentState := #instUnitModeStateManager.StateCurrent, history := #unitInterface.history)
   END_RUNG
   // the same network as SCL:
   "LUC_UpdateModeStateHistory"(currentMode := #instUnitModeStateManager.UnitModeCurrent,
                           currentState := #instUnitModeStateManager.StateCurrent,
                           history := #unitInterface.history);
END_REGION

REGION Network 18: Time Statistics
   // Determine the time that has been spend in modes and states.
   RUNG wire#powerrail
      #instUnitModeStateTimes(UnitModeCurrent := #instUnitModeStateManager.UnitModeCurrent, StateCurrent := #instUnitModeStateManager.StateCurrent, resetTimes :=, ModeTimeCurrent => #unitInterface.modeStateTimeStatistics.modeTimeCurrent, StateTimeCurrent => #unitInterface.modeStateTimeStatistics.stateTimeCurrent, AccTimeSinceReset => #unitInterface.modeStateTimeStatistics.accTimeSinceReset, actualTimeAllModes => #unitInterface.modeStateTimeStatistics.actualTimeAllModes, cumulativeTimeAllModes => #unitInterface.modeStateTimeStatistics.cumulativeTimeAllModes, actualTimeAllStatesOfAllModes => #unitInterface.modeStateTimeStatistics.actualTimeAllStatesOfAllModes, cumulativeTimeAllStatesOfAllModes => #unitInterface.modeStateTimeStatistics.cumulativeTimeAllStatesOfAllModes, actualTimeAllStatesOfCurrentMode => #unitInterface.modeStateTimeStatistics.actualTimeAllStatesOfCurrentMode, cumulativeTimeAllStatesOfCurrentMode => #unitInterface.modeStateTimeStatistics.cumulativeTimeAllStatesOfCurrentMode, cumulativeTimeCurrentMode => #unitInterface.modeStateTimeStatistics.cumulativeTimeCurrentMode)
   END_RUNG
   // the same network as SCL:
   #instUnitModeStateTimes(UnitModeCurrent := #instUnitModeStateManager.UnitModeCurrent,   // "LPMLV2022_UnitModeStateTimes"
                           StateCurrent := #instUnitModeStateManager.StateCurrent,
                           ModeTimeCurrent => #unitInterface.modeStateTimeStatistics.modeTimeCurrent,
                           StateTimeCurrent => #unitInterface.modeStateTimeStatistics.stateTimeCurrent,
                           AccTimeSinceReset => #unitInterface.modeStateTimeStatistics.accTimeSinceReset,
                           actualTimeAllModes => #unitInterface.modeStateTimeStatistics.actualTimeAllModes,
                           cumulativeTimeAllModes => #unitInterface.modeStateTimeStatistics.cumulativeTimeAllModes,
                           actualTimeAllStatesOfAllModes => #unitInterface.modeStateTimeStatistics.actualTimeAllStatesOfAllModes,
                           cumulativeTimeAllStatesOfAllModes => #unitInterface.modeStateTimeStatistics.cumulativeTimeAllStatesOfAllModes,
                           actualTimeAllStatesOfCurrentMode => #unitInterface.modeStateTimeStatistics.actualTimeAllStatesOfCurrentMode,
                           cumulativeTimeAllStatesOfCurrentMode => #unitInterface.modeStateTimeStatistics.cumulativeTimeAllStatesOfCurrentMode,
                           cumulativeTimeCurrentMode => #unitInterface.modeStateTimeStatistics.cumulativeTimeCurrentMode);
END_REGION

REGION Network 19: Stacklight
   // Determine light behaviour based on current mode and stacklight configuration
   RUNG wire#powerrail
      #instSignalStack(currentState := #instUnitModeStateManager.StateCurrent, freqClockBit := #globalStatus.clock.cycle1000Msec, disableHorn :=, hornPulseTime :=, processBypass :=, configuration := "Unit1.Config".signalStack, lightsByBool =>, lightsByDint =>, lightsByDWord => #unitInterface.signalStack, lightsStatus => "Unit1.EmNodes".signalStack)
   END_RUNG
   // the same network as SCL:
   #instSignalStack(currentState := #instUnitModeStateManager.StateCurrent,   // "LUC_SignalStack"
                    freqClockBit := #globalStatus.clock.cycle1000Msec,
                    configuration := "Unit1.Config".signalStack,
                    lightsByDWord => #unitInterface.signalStack,
                    lightsStatus => "Unit1.EmNodes".signalStack);
END_REGION

REGION Network 20: Stacklight Lamp
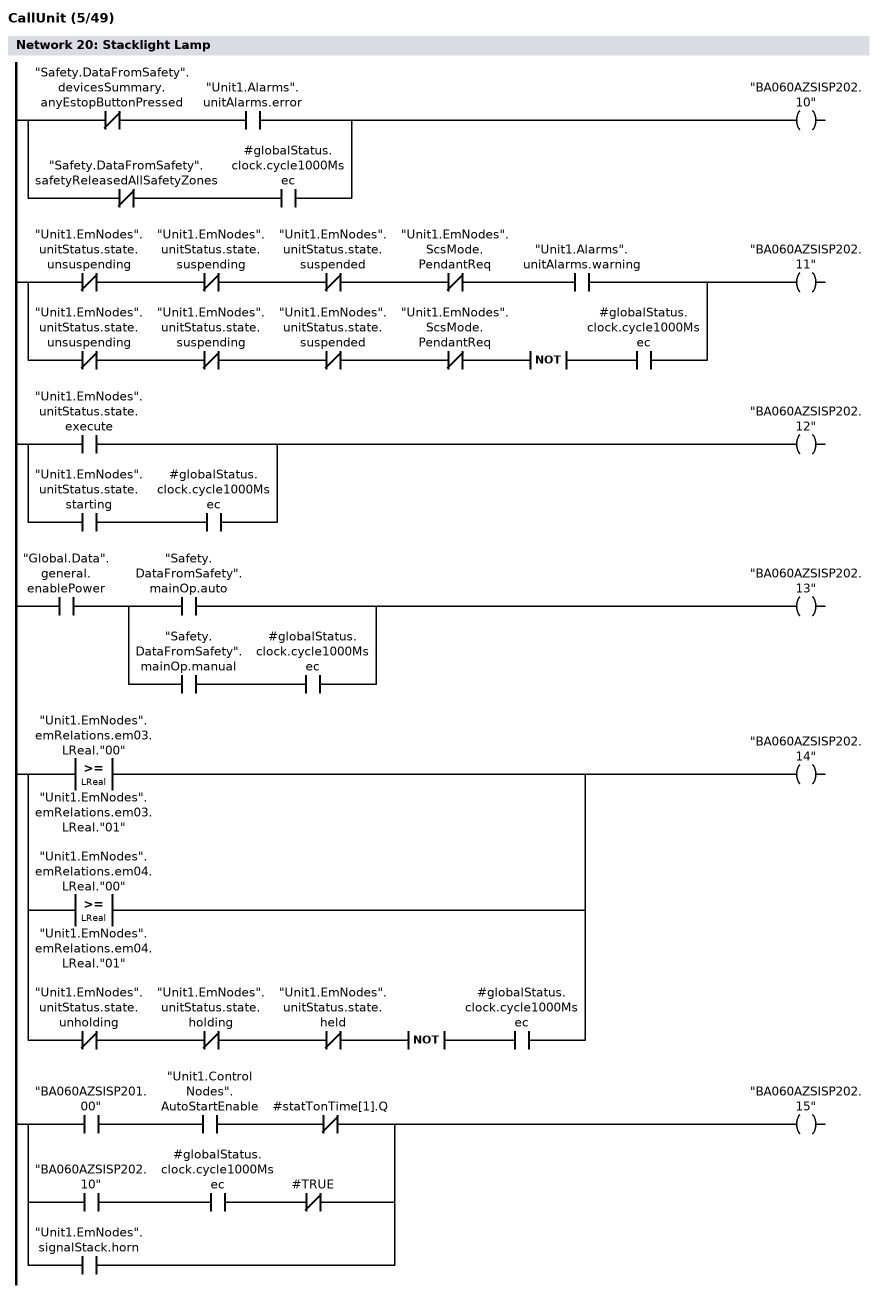
   RUNG wire#powerrail
      I_Contact( "Safety.DataFromSafety".devicesSummary.anyEstopButtonPressed )
      Contact( "Unit1.Alarms".unitAlarms.error )
      wire#w1
      Coil( "BA060AZSISP202.10" )
   END_RUNG
   RUNG wire#powerrail
      I_Contact( "Safety.DataFromSafety".safetyReleasedAllSafetyZones )
      Contact( #globalStatus.clock.cycle1000Msec )
   END_RUNG wire#w1
   RUNG wire#powerrail
      I_Contact( "Unit1.EmNodes".unitStatus.state.unsuspending )
      I_Contact( "Unit1.EmNodes".unitStatus.state.suspending )
      I_Contact( "Unit1.EmNodes".unitStatus.state.suspended )
      I_Contact( "Unit1.EmNodes".ScsMode.PendantReq )
      Contact( "Unit1.Alarms".unitAlarms.warning )
      wire#w2
      Coil( "BA060AZSISP202.11" )
   END_RUNG
   RUNG wire#powerrail
      I_Contact( "Unit1.EmNodes".unitStatus.state.unsuspending )
      I_Contact( "Unit1.EmNodes".unitStatus.state.suspending )
      I_Contact( "Unit1.EmNodes".unitStatus.state.suspended )
      I_Contact( "Unit1.EmNodes".ScsMode.PendantReq )
      Not()
      Contact( #globalStatus.clock.cycle1000Msec )
   END_RUNG wire#w2
   RUNG wire#powerrail
      Contact( "Unit1.EmNodes".unitStatus.state.execute )
      wire#w3
      Coil( "BA060AZSISP202.12" )
   END_RUNG
   RUNG wire#powerrail
      Contact( "Unit1.EmNodes".unitStatus.state.starting )
      Contact( #globalStatus.clock.cycle1000Msec )
   END_RUNG wire#w3
   RUNG wire#powerrail
      Contact( "Global.Data".general.enablePower )
      wire#w4
      Contact( "Safety.DataFromSafety".mainOp.auto )
      wire#w5
      Coil( "BA060AZSISP202.13" )
   END_RUNG
   RUNG wire#w4
      Contact( "Safety.DataFromSafety".mainOp.manual )
      Contact( #globalStatus.clock.cycle1000Msec )
   END_RUNG wire#w5
   RUNG wire#powerrail
      { S7_Templates := "SrcType := LReal" } GE_Contact(in1 := "Unit1.EmNodes".emRelations.em03.LReal."00", in2 := "Unit1.EmNodes".emRelations.em03.LReal."01")
      wire#w6
      Coil( "BA060AZSISP202.14" )
   END_RUNG
   RUNG wire#powerrail
      { S7_Templates := "SrcType := LReal" } GE_Contact(in1 := "Unit1.EmNodes".emRelations.em04.LReal."00", in2 := "Unit1.EmNodes".emRelations.em04.LReal."01")
   END_RUNG wire#w6
   RUNG wire#powerrail
      I_Contact( "Unit1.EmNodes".unitStatus.state.unholding )
      I_Contact( "Unit1.EmNodes".unitStatus.state.holding )
      I_Contact( "Unit1.EmNodes".unitStatus.state.held )
      Not()
      Contact( #globalStatus.clock.cycle1000Msec )
   END_RUNG wire#w6
   RUNG wire#powerrail
      Contact( "BA060AZSISP201.00" )
      Contact( "Unit1.ControlNodes".AutoStartEnable )
      I_Contact( #statTonTime[1].Q )
      wire#w7
      Coil( "BA060AZSISP202.15" )
   END_RUNG
   RUNG wire#powerrail
      Contact( "BA060AZSISP202.10" )
      Contact( #globalStatus.clock.cycle1000Msec )
      I_Contact( #TRUE )
   END_RUNG wire#w7
   RUNG wire#powerrail
      Contact( "Unit1.EmNodes".signalStack.horn )
   END_RUNG wire#w7
   // the same network as SCL:
   "BA060AZSISP202.10" := (NOT "Safety.DataFromSafety".devicesSummary.anyEstopButtonPressed AND "Unit1.Alarms".unitAlarms.error) OR (NOT "Safety.DataFromSafety".safetyReleasedAllSafetyZones AND #globalStatus.clock.cycle1000Msec);
   "BA060AZSISP202.11" := (NOT "Unit1.EmNodes".unitStatus.state.unsuspending AND NOT "Unit1.EmNodes".unitStatus.state.suspending AND NOT "Unit1.EmNodes".unitStatus.state.suspended AND NOT "Unit1.EmNodes".ScsMode.PendantReq AND "Unit1.Alarms".unitAlarms.warning) OR (NOT (NOT "Unit1.EmNodes".unitStatus.state.unsuspending AND NOT "Unit1.EmNodes".unitStatus.state.suspending AND NOT "Unit1.EmNodes".unitStatus.state.suspended AND NOT "Unit1.EmNodes".ScsMode.PendantReq) AND #globalStatus.clock.cycle1000Msec);
   "BA060AZSISP202.12" := "Unit1.EmNodes".unitStatus.state.execute OR ("Unit1.EmNodes".unitStatus.state.starting AND #globalStatus.clock.cycle1000Msec);
   "BA060AZSISP202.13" := "Global.Data".general.enablePower AND ("Safety.DataFromSafety".mainOp.auto OR ("Safety.DataFromSafety".mainOp.manual AND #globalStatus.clock.cycle1000Msec));
   "BA060AZSISP202.14" := ("Unit1.EmNodes".emRelations.em03.LReal."00" >= "Unit1.EmNodes".emRelations.em03.LReal."01") OR ("Unit1.EmNodes".emRelations.em04.LReal."00" >= "Unit1.EmNodes".emRelations.em04.LReal."01") OR (NOT (NOT "Unit1.EmNodes".unitStatus.state.unholding AND NOT "Unit1.EmNodes".unitStatus.state.holding AND NOT "Unit1.EmNodes".unitStatus.state.held) AND #globalStatus.clock.cycle1000Msec);
   "BA060AZSISP202.15" := ("BA060AZSISP201.00" AND "Unit1.ControlNodes".AutoStartEnable AND NOT #statTonTime[1].Q) OR ("BA060AZSISP202.10" AND #globalStatus.clock.cycle1000Msec AND NOT #TRUE) OR "Unit1.EmNodes".signalStack.horn;
END_REGION

REGION Network 21: QR Marker Stacklight Lamp
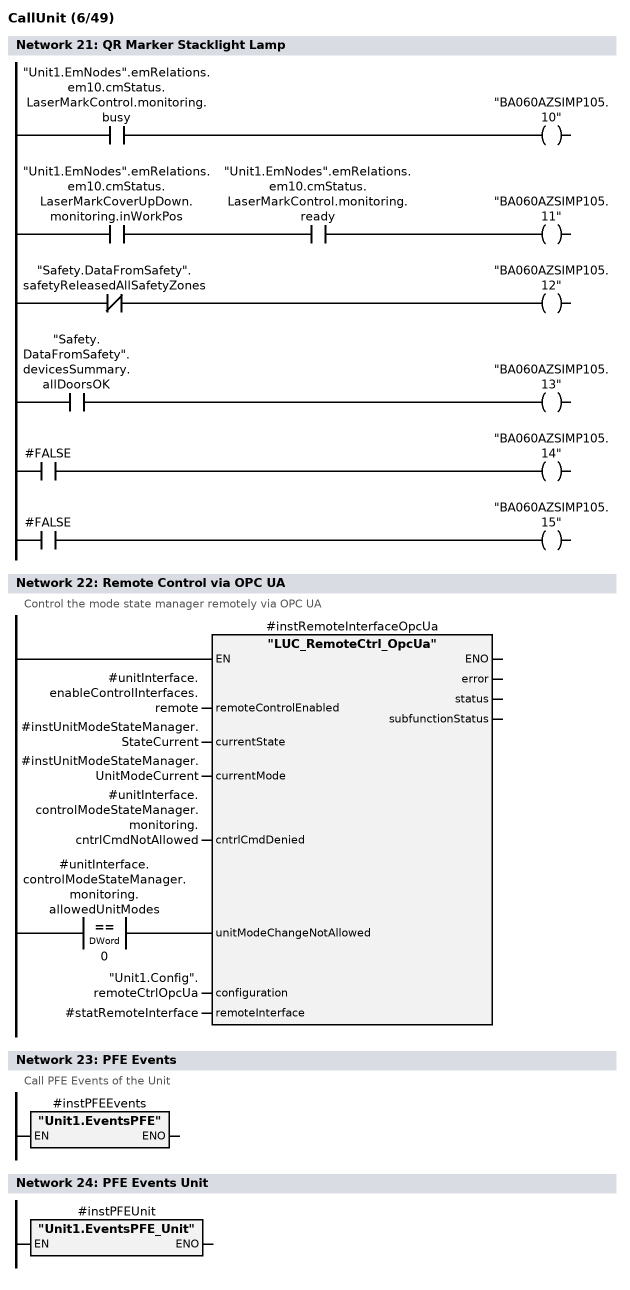
   RUNG wire#powerrail
      Contact( "Unit1.EmNodes".emRelations.em10.cmStatus.LaserMarkControl.monitoring.busy )
      Coil( "BA060AZSIMP105.10" )
   END_RUNG
   RUNG wire#powerrail
      Contact( "Unit1.EmNodes".emRelations.em10.cmStatus.LaserMarkCoverUpDown.monitoring.inWorkPos )
      Contact( "Unit1.EmNodes".emRelations.em10.cmStatus.LaserMarkControl.monitoring.ready )
      Coil( "BA060AZSIMP105.11" )
   END_RUNG
   RUNG wire#powerrail
      I_Contact( "Safety.DataFromSafety".safetyReleasedAllSafetyZones )
      Coil( "BA060AZSIMP105.12" )
   END_RUNG
   RUNG wire#powerrail
      Contact( "Safety.DataFromSafety".devicesSummary.allDoorsOK )
      Coil( "BA060AZSIMP105.13" )
   END_RUNG
   RUNG wire#powerrail
      Contact( #FALSE )
      Coil( "BA060AZSIMP105.14" )
   END_RUNG
   RUNG wire#powerrail
      Contact( #FALSE )
      Coil( "BA060AZSIMP105.15" )
   END_RUNG
   // the same network as SCL:
   "BA060AZSIMP105.10" := "Unit1.EmNodes".emRelations.em10.cmStatus.LaserMarkControl.monitoring.busy;
   "BA060AZSIMP105.11" := "Unit1.EmNodes".emRelations.em10.cmStatus.LaserMarkCoverUpDown.monitoring.inWorkPos AND "Unit1.EmNodes".emRelations.em10.cmStatus.LaserMarkControl.monitoring.ready;
   "BA060AZSIMP105.12" := NOT "Safety.DataFromSafety".safetyReleasedAllSafetyZones;
   "BA060AZSIMP105.13" := "Safety.DataFromSafety".devicesSummary.allDoorsOK;
   "BA060AZSIMP105.14" := #FALSE;
   "BA060AZSIMP105.15" := #FALSE;
END_REGION

REGION Network 22: Remote Control via OPC UA
   // Control the mode state manager remotely via OPC UA
   RUNG wire#powerrail
      #instRemoteInterfaceOpcUa(unitModeChangeNotAllowed := wire#w1, remoteControlEnabled := #unitInterface.enableControlInterfaces.remote, currentState := #instUnitModeStateManager.StateCurrent, currentMode := #instUnitModeStateManager.UnitModeCurrent, cntrlCmdDenied := #unitInterface.controlModeStateManager.monitoring.cntrlCmdNotAllowed, configuration := "Unit1.Config".remoteCtrlOpcUa, remoteInterface := #statRemoteInterface, error =>, status =>, subfunctionStatus =>)
   END_RUNG
   RUNG wire#powerrail
      { S7_Templates := "SrcType := DWord" } EQ_Contact(in1 := #unitInterface.controlModeStateManager.monitoring.allowedUnitModes, in2 := 0)
   END_RUNG wire#w1
   // the same network as SCL:
   #instRemoteInterfaceOpcUa(remoteControlEnabled := #unitInterface.enableControlInterfaces.remote,   // "LUC_RemoteCtrl_OpcUa"
                           currentState := #instUnitModeStateManager.StateCurrent,
                           currentMode := #instUnitModeStateManager.UnitModeCurrent,
                           cntrlCmdDenied := #unitInterface.controlModeStateManager.monitoring.cntrlCmdNotAllowed,
                           unitModeChangeNotAllowed := #unitInterface.controlModeStateManager.monitoring.allowedUnitModes = 0,
                           configuration := "Unit1.Config".remoteCtrlOpcUa,
                           remoteInterface := #statRemoteInterface);
END_REGION

REGION Network 23: PFE Events
   // Call PFE Events of the Unit
   RUNG wire#powerrail
      #instPFEEvents()
   END_RUNG
   // the same network as SCL:
   #instPFEEvents();   // "Unit1.EventsPFE"
END_REGION

REGION Network 24: PFE Events Unit
   RUNG wire#powerrail
      #instPFEUnit()
   END_RUNG
   // the same network as SCL:
   #instPFEUnit();   // "Unit1.EventsPFE_Unit"
END_REGION

REGION Network 25: Clock Memory
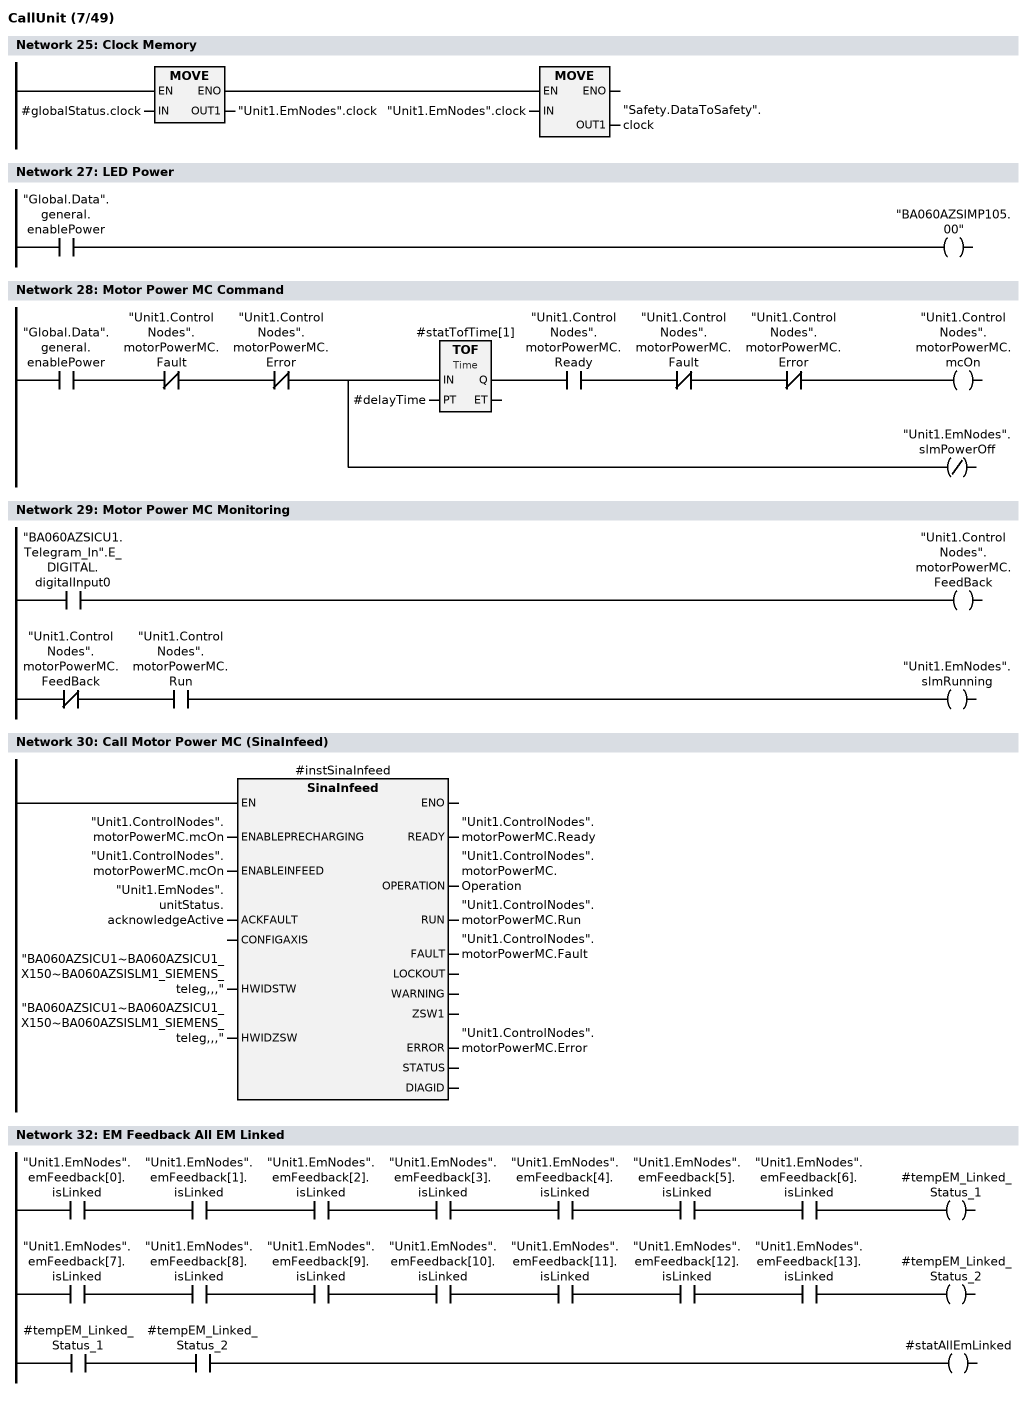
   RUNG wire#powerrail
      Move(in := #globalStatus.clock, out1 => "Unit1.EmNodes".clock)
      Move(in := "Unit1.EmNodes".clock, out1 => "Safety.DataToSafety".clock)
   END_RUNG
   // the same network as SCL:
   "Unit1.EmNodes".clock := #globalStatus.clock;
   "Safety.DataToSafety".clock := "Unit1.EmNodes".clock;
END_REGION

REGION Network 26: ******************** Power ********************
END_REGION

REGION Network 27: LED Power
   RUNG wire#powerrail
      Contact( "Global.Data".general.enablePower )
      Coil( "BA060AZSIMP105.00" )
   END_RUNG
   // the same network as SCL:
   "BA060AZSIMP105.00" := "Global.Data".general.enablePower;
END_REGION

REGION Network 28: Motor Power MC Command
   RUNG wire#powerrail
      Contact( "Global.Data".general.enablePower )
      I_Contact( "Unit1.ControlNodes".motorPowerMC.Fault )
      I_Contact( "Unit1.ControlNodes".motorPowerMC.Error )
      wire#w1
      { S7_Templates := "time_type := Time" } #statTofTime[1].TOF(pt := #delayTime, et =>)
      Contact( "Unit1.ControlNodes".motorPowerMC.Ready )
      I_Contact( "Unit1.ControlNodes".motorPowerMC.Fault )
      I_Contact( "Unit1.ControlNodes".motorPowerMC.Error )
      Coil( "Unit1.ControlNodes".motorPowerMC.mcOn )
   END_RUNG
   RUNG wire#w1
      I_Coil( "Unit1.EmNodes".slmPowerOff )
   END_RUNG
   // the same network as SCL:
   #_w1 := "Global.Data".general.enablePower AND NOT "Unit1.ControlNodes".motorPowerMC.Fault AND NOT "Unit1.ControlNodes".motorPowerMC.Error;
   #statTofTime[1].TOF(IN := #_w1, PT := #delayTime);
   "Unit1.ControlNodes".motorPowerMC.mcOn := #statTofTime[1].Q AND "Unit1.ControlNodes".motorPowerMC.Ready AND NOT "Unit1.ControlNodes".motorPowerMC.Fault AND NOT "Unit1.ControlNodes".motorPowerMC.Error;
   "Unit1.EmNodes".slmPowerOff := NOT #_w1;
END_REGION

REGION Network 29: Motor Power MC Monitoring
   RUNG wire#powerrail
      Contact( "BA060AZSICU1.Telegram_In".E_DIGITAL.digitalInput0 )
      Coil( "Unit1.ControlNodes".motorPowerMC.FeedBack )
   END_RUNG
   RUNG wire#powerrail
      I_Contact( "Unit1.ControlNodes".motorPowerMC.FeedBack )
      Contact( "Unit1.ControlNodes".motorPowerMC.Run )
      Coil( "Unit1.EmNodes".slmRunning )
   END_RUNG
   // the same network as SCL:
   "Unit1.ControlNodes".motorPowerMC.FeedBack := "BA060AZSICU1.Telegram_In".E_DIGITAL.digitalInput0;
   "Unit1.EmNodes".slmRunning := NOT "Unit1.ControlNodes".motorPowerMC.FeedBack AND "Unit1.ControlNodes".motorPowerMC.Run;
END_REGION

REGION Network 30: Call Motor Power MC (SinaInfeed)
   RUNG wire#powerrail
      #instSinaInfeed.SinaInfeed(EnablePrecharging := "Unit1.ControlNodes".motorPowerMC.mcOn, EnableInfeed := "Unit1.ControlNodes".motorPowerMC.mcOn, AckFault := "Unit1.EmNodes".unitStatus.acknowledgeActive, ConfigAxis :=, HWIDSTW := "BA060AZSICU1~BA060AZSICU1_X150~BA060AZSISLM1_SIEMENS_teleg,,,", HWIDZSW := "BA060AZSICU1~BA060AZSICU1_X150~BA060AZSISLM1_SIEMENS_teleg,,,", Ready => "Unit1.ControlNodes".motorPowerMC.Ready, Operation => "Unit1.ControlNodes".motorPowerMC.Operation, Run => "Unit1.ControlNodes".motorPowerMC.Run, Fault => "Unit1.ControlNodes".motorPowerMC.Fault, Lockout =>, Warning =>, ZSW1 =>, Error => "Unit1.ControlNodes".motorPowerMC.Error, Status =>, DiagID =>)
   END_RUNG
   // the same network as SCL:
   #instSinaInfeed(EnablePrecharging := "Unit1.ControlNodes".motorPowerMC.mcOn,   // SinaInfeed
                   EnableInfeed := "Unit1.ControlNodes".motorPowerMC.mcOn,
                   AckFault := "Unit1.EmNodes".unitStatus.acknowledgeActive,
                   HWIDSTW := "BA060AZSICU1~BA060AZSICU1_X150~BA060AZSISLM1_SIEMENS_teleg,,,",
                   HWIDZSW := "BA060AZSICU1~BA060AZSICU1_X150~BA060AZSISLM1_SIEMENS_teleg,,,",
                   Ready => "Unit1.ControlNodes".motorPowerMC.Ready,
                   Operation => "Unit1.ControlNodes".motorPowerMC.Operation,
                   Run => "Unit1.ControlNodes".motorPowerMC.Run,
                   Fault => "Unit1.ControlNodes".motorPowerMC.Fault,
                   Error => "Unit1.ControlNodes".motorPowerMC.Error);
END_REGION

REGION Network 31: ******************** Local Operation Box ********************
END_REGION

REGION Network 32: EM Feedback All EM Linked
   RUNG wire#powerrail
      Contact( "Unit1.EmNodes".emFeedback[0].isLinked )
      Contact( "Unit1.EmNodes".emFeedback[1].isLinked )
      Contact( "Unit1.EmNodes".emFeedback[2].isLinked )
      Contact( "Unit1.EmNodes".emFeedback[3].isLinked )
      Contact( "Unit1.EmNodes".emFeedback[4].isLinked )
      Contact( "Unit1.EmNodes".emFeedback[5].isLinked )
      Contact( "Unit1.EmNodes".emFeedback[6].isLinked )
      Coil( #tempEM_Linked_Status_1 )
   END_RUNG
   RUNG wire#powerrail
      Contact( "Unit1.EmNodes".emFeedback[7].isLinked )
      Contact( "Unit1.EmNodes".emFeedback[8].isLinked )
      Contact( "Unit1.EmNodes".emFeedback[9].isLinked )
      Contact( "Unit1.EmNodes".emFeedback[10].isLinked )
      Contact( "Unit1.EmNodes".emFeedback[11].isLinked )
      Contact( "Unit1.EmNodes".emFeedback[12].isLinked )
      Contact( "Unit1.EmNodes".emFeedback[13].isLinked )
      Coil( #tempEM_Linked_Status_2 )
   END_RUNG
   RUNG wire#powerrail
      Contact( #tempEM_Linked_Status_1 )
      Contact( #tempEM_Linked_Status_2 )
      Coil( #statAllEmLinked )
   END_RUNG
   // the same network as SCL:
   #tempEM_Linked_Status_1 := "Unit1.EmNodes".emFeedback[0].isLinked AND "Unit1.EmNodes".emFeedback[1].isLinked AND "Unit1.EmNodes".emFeedback[2].isLinked AND "Unit1.EmNodes".emFeedback[3].isLinked AND "Unit1.EmNodes".emFeedback[4].isLinked AND "Unit1.EmNodes".emFeedback[5].isLinked AND "Unit1.EmNodes".emFeedback[6].isLinked;
   #tempEM_Linked_Status_2 := "Unit1.EmNodes".emFeedback[7].isLinked AND "Unit1.EmNodes".emFeedback[8].isLinked AND "Unit1.EmNodes".emFeedback[9].isLinked AND "Unit1.EmNodes".emFeedback[10].isLinked AND "Unit1.EmNodes".emFeedback[11].isLinked AND "Unit1.EmNodes".emFeedback[12].isLinked AND "Unit1.EmNodes".emFeedback[13].isLinked;
   #statAllEmLinked := #tempEM_Linked_Status_1 AND #tempEM_Linked_Status_2;
END_REGION

REGION Network 33: Enable interfaces to control the unit
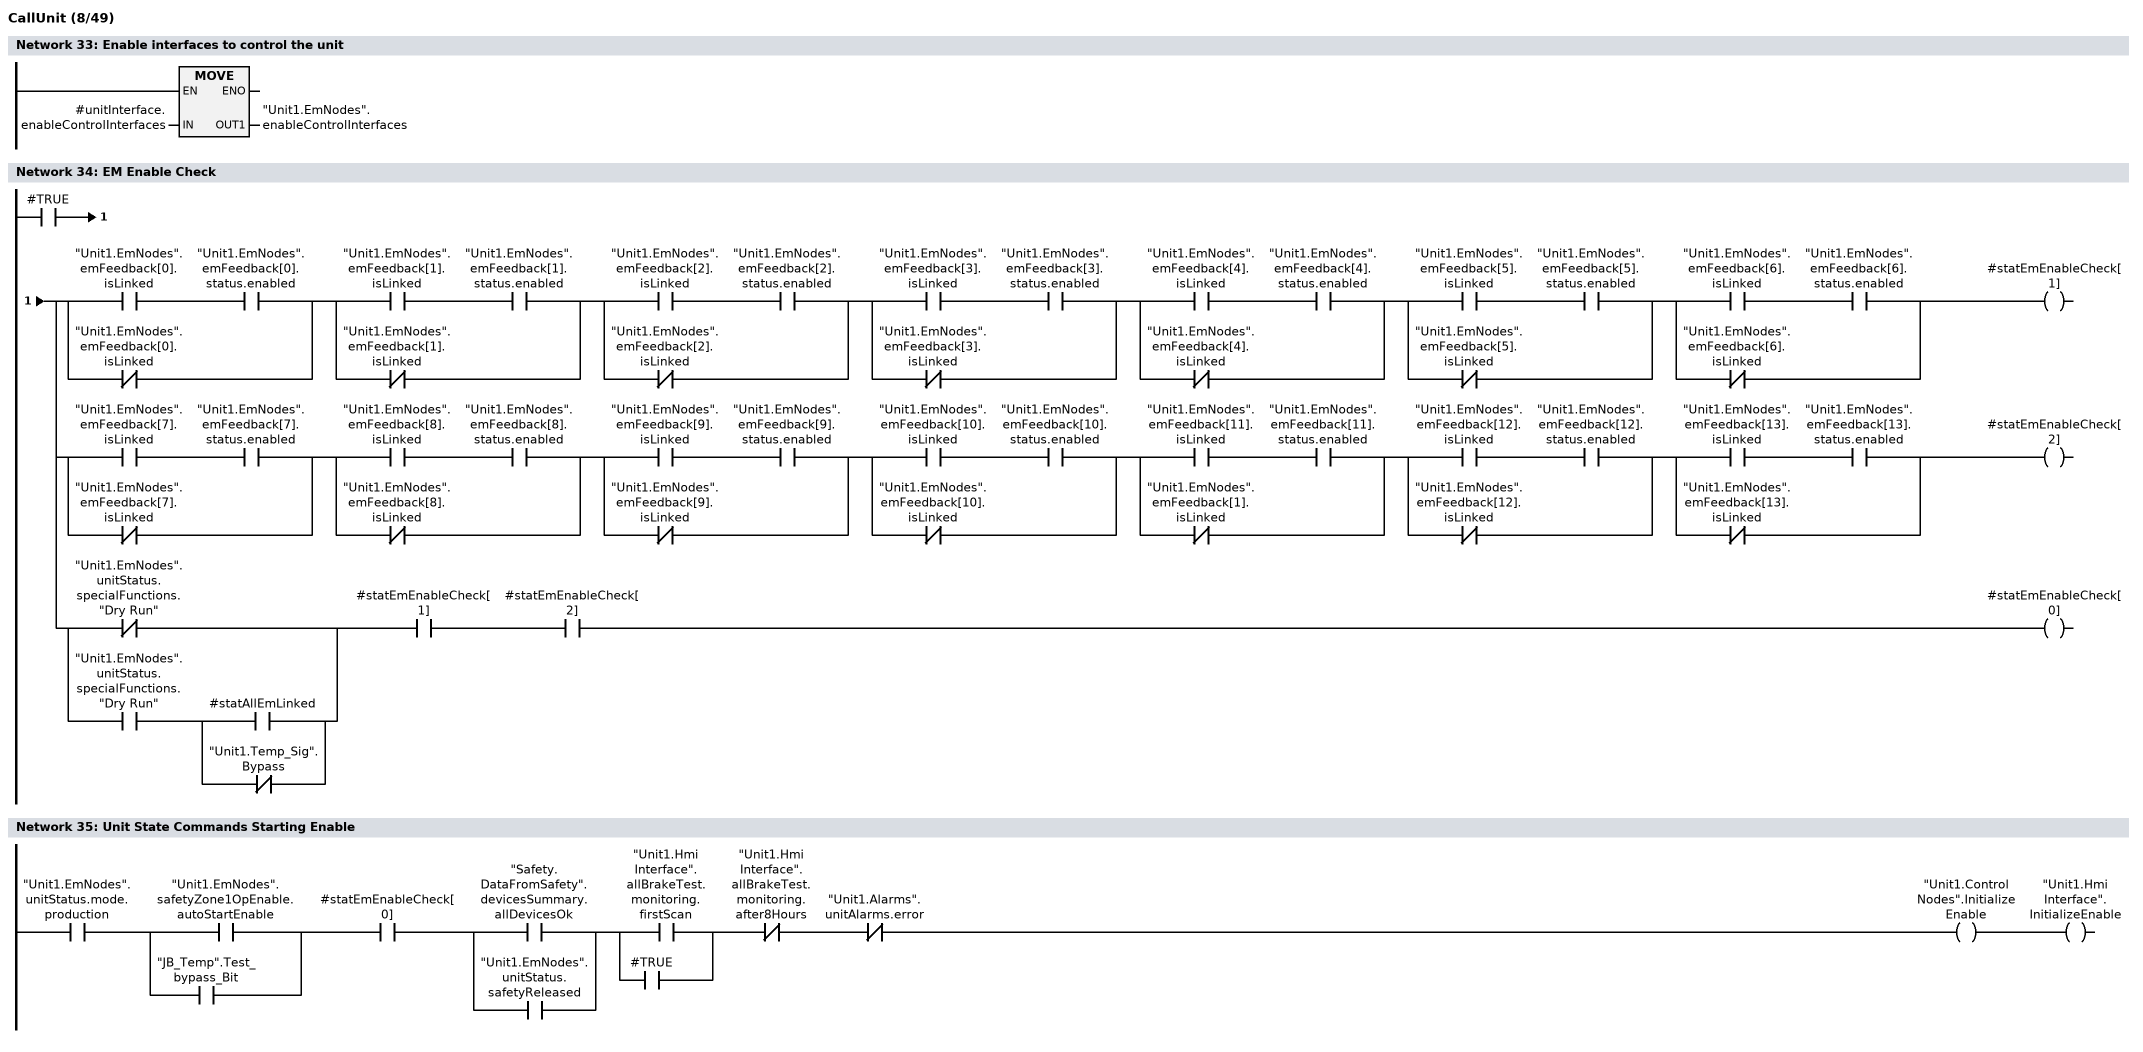
   RUNG wire#powerrail
      Move(in := #unitInterface.enableControlInterfaces, out1 => "Unit1.EmNodes".enableControlInterfaces)
   END_RUNG
   // the same network as SCL:
   "Unit1.EmNodes".enableControlInterfaces := #unitInterface.enableControlInterfaces;
END_REGION

REGION Network 34: EM Enable Check
   RUNG wire#powerrail
      Contact( #TRUE )
      wire#w1
      Contact( "Unit1.EmNodes".emFeedback[0].isLinked )
      Contact( "Unit1.EmNodes".emFeedback[0].status.enabled )
      wire#w2
      Contact( "Unit1.EmNodes".emFeedback[1].isLinked )
      Contact( "Unit1.EmNodes".emFeedback[1].status.enabled )
      wire#w3
      Contact( "Unit1.EmNodes".emFeedback[2].isLinked )
      Contact( "Unit1.EmNodes".emFeedback[2].status.enabled )
      wire#w4
      Contact( "Unit1.EmNodes".emFeedback[3].isLinked )
      Contact( "Unit1.EmNodes".emFeedback[3].status.enabled )
      wire#w5
      Contact( "Unit1.EmNodes".emFeedback[4].isLinked )
      Contact( "Unit1.EmNodes".emFeedback[4].status.enabled )
      wire#w6
      Contact( "Unit1.EmNodes".emFeedback[5].isLinked )
      Contact( "Unit1.EmNodes".emFeedback[5].status.enabled )
      wire#w7
      Contact( "Unit1.EmNodes".emFeedback[6].isLinked )
      Contact( "Unit1.EmNodes".emFeedback[6].status.enabled )
      wire#w8
      Coil( #statEmEnableCheck[1] )
   END_RUNG
   RUNG wire#w1
      I_Contact( "Unit1.EmNodes".emFeedback[0].isLinked )
   END_RUNG wire#w2
   RUNG wire#w2
      I_Contact( "Unit1.EmNodes".emFeedback[1].isLinked )
   END_RUNG wire#w3
   RUNG wire#w3
      I_Contact( "Unit1.EmNodes".emFeedback[2].isLinked )
   END_RUNG wire#w4
   RUNG wire#w4
      I_Contact( "Unit1.EmNodes".emFeedback[3].isLinked )
   END_RUNG wire#w5
   RUNG wire#w5
      I_Contact( "Unit1.EmNodes".emFeedback[4].isLinked )
   END_RUNG wire#w6
   RUNG wire#w6
      I_Contact( "Unit1.EmNodes".emFeedback[5].isLinked )
   END_RUNG wire#w7
   RUNG wire#w7
      I_Contact( "Unit1.EmNodes".emFeedback[6].isLinked )
   END_RUNG wire#w8
   RUNG wire#w1
      Contact( "Unit1.EmNodes".emFeedback[7].isLinked )
      Contact( "Unit1.EmNodes".emFeedback[7].status.enabled )
      wire#w9
      Contact( "Unit1.EmNodes".emFeedback[8].isLinked )
      Contact( "Unit1.EmNodes".emFeedback[8].status.enabled )
      wire#w10
      Contact( "Unit1.EmNodes".emFeedback[9].isLinked )
      Contact( "Unit1.EmNodes".emFeedback[9].status.enabled )
      wire#w11
      Contact( "Unit1.EmNodes".emFeedback[10].isLinked )
      Contact( "Unit1.EmNodes".emFeedback[10].status.enabled )
      wire#w12
      Contact( "Unit1.EmNodes".emFeedback[11].isLinked )
      Contact( "Unit1.EmNodes".emFeedback[11].status.enabled )
      wire#w13
      Contact( "Unit1.EmNodes".emFeedback[12].isLinked )
      Contact( "Unit1.EmNodes".emFeedback[12].status.enabled )
      wire#w14
      Contact( "Unit1.EmNodes".emFeedback[13].isLinked )
      Contact( "Unit1.EmNodes".emFeedback[13].status.enabled )
      wire#w15
      Coil( #statEmEnableCheck[2] )
   END_RUNG
   RUNG wire#w1
      I_Contact( "Unit1.EmNodes".emFeedback[7].isLinked )
   END_RUNG wire#w9
   RUNG wire#w9
      I_Contact( "Unit1.EmNodes".emFeedback[8].isLinked )
   END_RUNG wire#w10
   RUNG wire#w10
      I_Contact( "Unit1.EmNodes".emFeedback[9].isLinked )
   END_RUNG wire#w11
   RUNG wire#w11
      I_Contact( "Unit1.EmNodes".emFeedback[10].isLinked )
   END_RUNG wire#w12
   RUNG wire#w12
      I_Contact( "Unit1.EmNodes".emFeedback[1].isLinked )
   END_RUNG wire#w13
   RUNG wire#w13
      I_Contact( "Unit1.EmNodes".emFeedback[12].isLinked )
   END_RUNG wire#w14
   RUNG wire#w14
      I_Contact( "Unit1.EmNodes".emFeedback[13].isLinked )
   END_RUNG wire#w15
   RUNG wire#w1
      I_Contact( "Unit1.EmNodes".unitStatus.specialFunctions."Dry Run" )
      wire#w16
      Contact( #statEmEnableCheck[1] )
      Contact( #statEmEnableCheck[2] )
      Coil( #statEmEnableCheck[0] )
   END_RUNG
   RUNG wire#w1
      Contact( "Unit1.EmNodes".unitStatus.specialFunctions."Dry Run" )
      wire#w17
      Contact( #statAllEmLinked )
   END_RUNG wire#w16
   RUNG wire#w17
      I_Contact( "Unit1.Temp_Sig".Bypass )
   END_RUNG wire#w16
   // the same network as SCL:
   #statEmEnableCheck[1] := #TRUE AND (("Unit1.EmNodes".emFeedback[0].isLinked AND "Unit1.EmNodes".emFeedback[0].status.enabled) OR NOT "Unit1.EmNodes".emFeedback[0].isLinked) AND (("Unit1.EmNodes".emFeedback[1].isLinked AND "Unit1.EmNodes".emFeedback[1].status.enabled) OR NOT "Unit1.EmNodes".emFeedback[1].isLinked) AND (("Unit1.EmNodes".emFeedback[2].isLinked AND "Unit1.EmNodes".emFeedback[2].status.enabled) OR NOT "Unit1.EmNodes".emFeedback[2].isLinked) AND (("Unit1.EmNodes".emFeedback[3].isLinked AND "Unit1.EmNodes".emFeedback[3].status.enabled) OR NOT "Unit1.EmNodes".emFeedback[3].isLinked) AND (("Unit1.EmNodes".emFeedback[4].isLinked AND "Unit1.EmNodes".emFeedback[4].status.enabled) OR NOT "Unit1.EmNodes".emFeedback[4].isLinked) AND (("Unit1.EmNodes".emFeedback[5].isLinked AND "Unit1.EmNodes".emFeedback[5].status.enabled) OR NOT "Unit1.EmNodes".emFeedback[5].isLinked) AND (("Unit1.EmNodes".emFeedback[6].isLinked AND "Unit1.EmNodes".emFeedback[6].status.enabled) OR NOT "Unit1.EmNodes".emFeedback[6].isLinked);
   #statEmEnableCheck[2] := #TRUE AND (("Unit1.EmNodes".emFeedback[7].isLinked AND "Unit1.EmNodes".emFeedback[7].status.enabled) OR NOT "Unit1.EmNodes".emFeedback[7].isLinked) AND (("Unit1.EmNodes".emFeedback[8].isLinked AND "Unit1.EmNodes".emFeedback[8].status.enabled) OR NOT "Unit1.EmNodes".emFeedback[8].isLinked) AND (("Unit1.EmNodes".emFeedback[9].isLinked AND "Unit1.EmNodes".emFeedback[9].status.enabled) OR NOT "Unit1.EmNodes".emFeedback[9].isLinked) AND (("Unit1.EmNodes".emFeedback[10].isLinked AND "Unit1.EmNodes".emFeedback[10].status.enabled) OR NOT "Unit1.EmNodes".emFeedback[10].isLinked) AND (("Unit1.EmNodes".emFeedback[11].isLinked AND "Unit1.EmNodes".emFeedback[11].status.enabled) OR NOT "Unit1.EmNodes".emFeedback[1].isLinked) AND (("Unit1.EmNodes".emFeedback[12].isLinked AND "Unit1.EmNodes".emFeedback[12].status.enabled) OR NOT "Unit1.EmNodes".emFeedback[12].isLinked) AND (("Unit1.EmNodes".emFeedback[13].isLinked AND "Unit1.EmNodes".emFeedback[13].status.enabled) OR NOT "Unit1.EmNodes".emFeedback[13].isLinked);
   #statEmEnableCheck[0] := #TRUE AND (NOT "Unit1.EmNodes".unitStatus.specialFunctions."Dry Run" OR ("Unit1.EmNodes".unitStatus.specialFunctions."Dry Run" AND (#statAllEmLinked OR NOT "Unit1.Temp_Sig".Bypass))) AND #statEmEnableCheck[1] AND #statEmEnableCheck[2];
END_REGION

REGION Network 35: Unit State Commands Starting Enable
   RUNG wire#powerrail
      Contact( "Unit1.EmNodes".unitStatus.mode.production )
      wire#w1
      Contact( "Unit1.EmNodes".safetyZone1OpEnable.autoStartEnable )
      wire#w2
      Contact( #statEmEnableCheck[0] )
      wire#w3
      Contact( "Safety.DataFromSafety".devicesSummary.allDevicesOk )
      wire#w4
      Contact( "Unit1.HmiInterface".allBrakeTest.monitoring.firstScan )
      wire#w5
      I_Contact( "Unit1.HmiInterface".allBrakeTest.monitoring.after8Hours )
      I_Contact( "Unit1.Alarms".unitAlarms.error )
      Coil( "Unit1.ControlNodes".InitializeEnable )
      Coil( "Unit1.HmiInterface".InitializeEnable )
   END_RUNG
   RUNG wire#w1
      Contact( "JB_Temp".Test_bypass_Bit )
   END_RUNG wire#w2
   RUNG wire#w3
      Contact( "Unit1.EmNodes".unitStatus.safetyReleased )
   END_RUNG wire#w4
   RUNG wire#w4
      Contact( #TRUE )
   END_RUNG wire#w5
   // the same network as SCL:
   "Unit1.ControlNodes".InitializeEnable := "Unit1.EmNodes".unitStatus.mode.production AND ("Unit1.EmNodes".safetyZone1OpEnable.autoStartEnable OR "JB_Temp".Test_bypass_Bit) AND #statEmEnableCheck[0] AND ("Safety.DataFromSafety".devicesSummary.allDevicesOk OR "Unit1.EmNodes".unitStatus.safetyReleased) AND ("Unit1.HmiInterface".allBrakeTest.monitoring.firstScan OR #TRUE) AND NOT "Unit1.HmiInterface".allBrakeTest.monitoring.after8Hours AND NOT "Unit1.Alarms".unitAlarms.error;
   "Unit1.HmiInterface".InitializeEnable := "Unit1.ControlNodes".InitializeEnable;
END_REGION

REGION Network 36: EM initialized + Homed Check
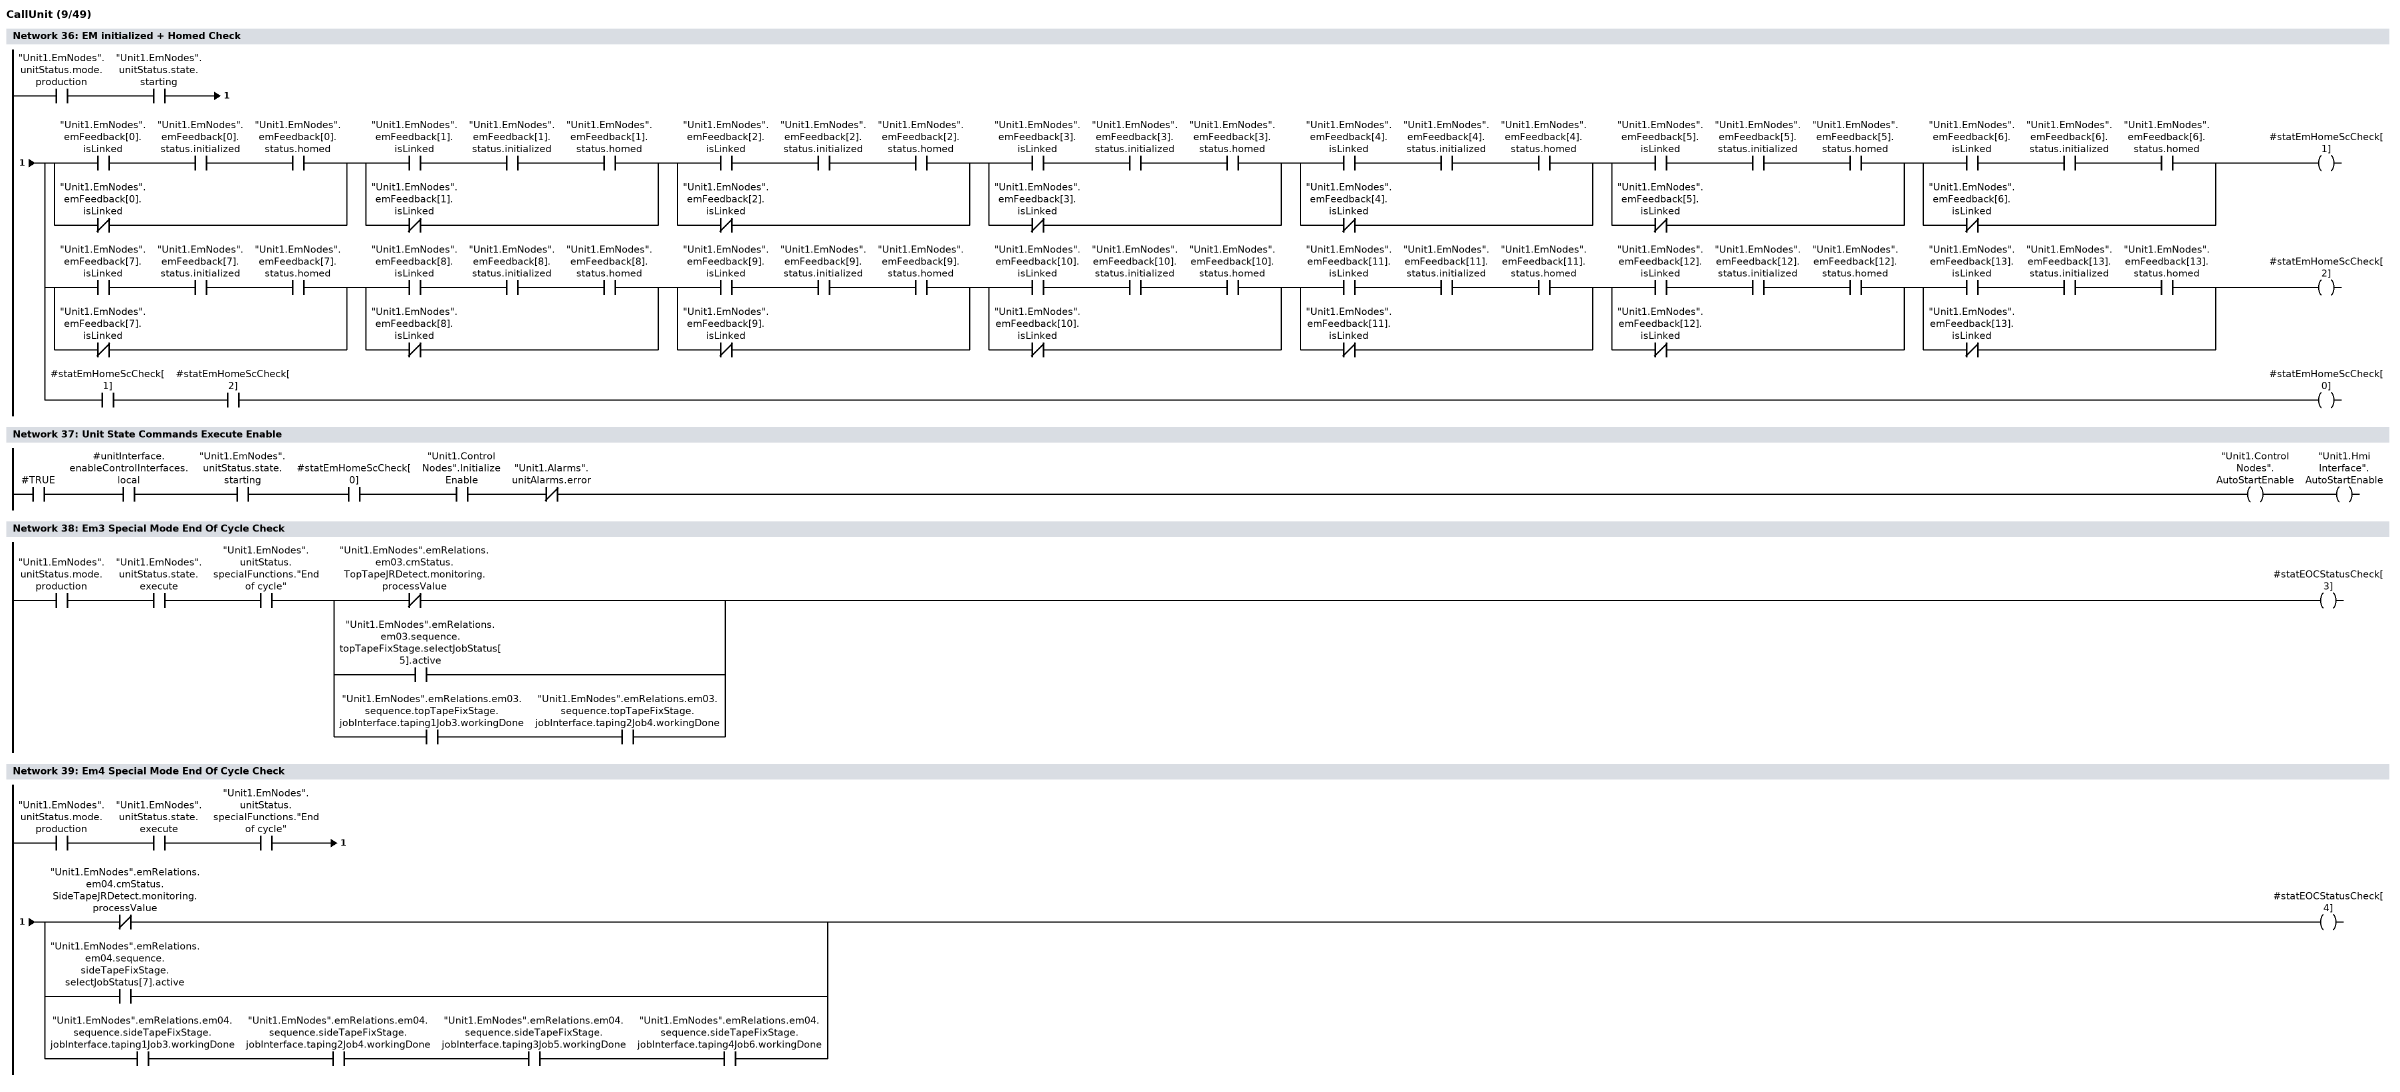
   RUNG wire#powerrail
      Contact( "Unit1.EmNodes".unitStatus.mode.production )
      Contact( "Unit1.EmNodes".unitStatus.state.starting )
      wire#w1
      Contact( "Unit1.EmNodes".emFeedback[0].isLinked )
      Contact( "Unit1.EmNodes".emFeedback[0].status.initialized )
      Contact( "Unit1.EmNodes".emFeedback[0].status.homed )
      wire#w2
      Contact( "Unit1.EmNodes".emFeedback[1].isLinked )
      Contact( "Unit1.EmNodes".emFeedback[1].status.initialized )
      Contact( "Unit1.EmNodes".emFeedback[1].status.homed )
      wire#w3
      Contact( "Unit1.EmNodes".emFeedback[2].isLinked )
      Contact( "Unit1.EmNodes".emFeedback[2].status.initialized )
      Contact( "Unit1.EmNodes".emFeedback[2].status.homed )
      wire#w4
      Contact( "Unit1.EmNodes".emFeedback[3].isLinked )
      Contact( "Unit1.EmNodes".emFeedback[3].status.initialized )
      Contact( "Unit1.EmNodes".emFeedback[3].status.homed )
      wire#w5
      Contact( "Unit1.EmNodes".emFeedback[4].isLinked )
      Contact( "Unit1.EmNodes".emFeedback[4].status.initialized )
      Contact( "Unit1.EmNodes".emFeedback[4].status.homed )
      wire#w6
      Contact( "Unit1.EmNodes".emFeedback[5].isLinked )
      Contact( "Unit1.EmNodes".emFeedback[5].status.initialized )
      Contact( "Unit1.EmNodes".emFeedback[5].status.homed )
      wire#w7
      Contact( "Unit1.EmNodes".emFeedback[6].isLinked )
      Contact( "Unit1.EmNodes".emFeedback[6].status.initialized )
      Contact( "Unit1.EmNodes".emFeedback[6].status.homed )
      wire#w8
      Coil( #statEmHomeScCheck[1] )
   END_RUNG
   RUNG wire#w1
      I_Contact( "Unit1.EmNodes".emFeedback[0].isLinked )
   END_RUNG wire#w2
   RUNG wire#w2
      I_Contact( "Unit1.EmNodes".emFeedback[1].isLinked )
   END_RUNG wire#w3
   RUNG wire#w3
      I_Contact( "Unit1.EmNodes".emFeedback[2].isLinked )
   END_RUNG wire#w4
   RUNG wire#w4
      I_Contact( "Unit1.EmNodes".emFeedback[3].isLinked )
   END_RUNG wire#w5
   RUNG wire#w5
      I_Contact( "Unit1.EmNodes".emFeedback[4].isLinked )
   END_RUNG wire#w6
   RUNG wire#w6
      I_Contact( "Unit1.EmNodes".emFeedback[5].isLinked )
   END_RUNG wire#w7
   RUNG wire#w7
      I_Contact( "Unit1.EmNodes".emFeedback[6].isLinked )
   END_RUNG wire#w8
   RUNG wire#w1
      Contact( "Unit1.EmNodes".emFeedback[7].isLinked )
      Contact( "Unit1.EmNodes".emFeedback[7].status.initialized )
      Contact( "Unit1.EmNodes".emFeedback[7].status.homed )
      wire#w9
      Contact( "Unit1.EmNodes".emFeedback[8].isLinked )
      Contact( "Unit1.EmNodes".emFeedback[8].status.initialized )
      Contact( "Unit1.EmNodes".emFeedback[8].status.homed )
      wire#w10
      Contact( "Unit1.EmNodes".emFeedback[9].isLinked )
      Contact( "Unit1.EmNodes".emFeedback[9].status.initialized )
      Contact( "Unit1.EmNodes".emFeedback[9].status.homed )
      wire#w11
      Contact( "Unit1.EmNodes".emFeedback[10].isLinked )
      Contact( "Unit1.EmNodes".emFeedback[10].status.initialized )
      Contact( "Unit1.EmNodes".emFeedback[10].status.homed )
      wire#w12
      Contact( "Unit1.EmNodes".emFeedback[11].isLinked )
      Contact( "Unit1.EmNodes".emFeedback[11].status.initialized )
      Contact( "Unit1.EmNodes".emFeedback[11].status.homed )
      wire#w13
      Contact( "Unit1.EmNodes".emFeedback[12].isLinked )
      Contact( "Unit1.EmNodes".emFeedback[12].status.initialized )
      Contact( "Unit1.EmNodes".emFeedback[12].status.homed )
      wire#w14
      Contact( "Unit1.EmNodes".emFeedback[13].isLinked )
      Contact( "Unit1.EmNodes".emFeedback[13].status.initialized )
      Contact( "Unit1.EmNodes".emFeedback[13].status.homed )
      wire#w15
      Coil( #statEmHomeScCheck[2] )
   END_RUNG
   RUNG wire#w1
      I_Contact( "Unit1.EmNodes".emFeedback[7].isLinked )
   END_RUNG wire#w9
   RUNG wire#w9
      I_Contact( "Unit1.EmNodes".emFeedback[8].isLinked )
   END_RUNG wire#w10
   RUNG wire#w10
      I_Contact( "Unit1.EmNodes".emFeedback[9].isLinked )
   END_RUNG wire#w11
   RUNG wire#w11
      I_Contact( "Unit1.EmNodes".emFeedback[10].isLinked )
   END_RUNG wire#w12
   RUNG wire#w12
      I_Contact( "Unit1.EmNodes".emFeedback[11].isLinked )
   END_RUNG wire#w13
   RUNG wire#w13
      I_Contact( "Unit1.EmNodes".emFeedback[12].isLinked )
   END_RUNG wire#w14
   RUNG wire#w14
      I_Contact( "Unit1.EmNodes".emFeedback[13].isLinked )
   END_RUNG wire#w15
   RUNG wire#w1
      Contact( #statEmHomeScCheck[1] )
      Contact( #statEmHomeScCheck[2] )
      Coil( #statEmHomeScCheck[0] )
   END_RUNG
   // the same network as SCL:
   #_w1 := "Unit1.EmNodes".unitStatus.mode.production AND "Unit1.EmNodes".unitStatus.state.starting;
   #statEmHomeScCheck[1] := #_w1 AND (("Unit1.EmNodes".emFeedback[0].isLinked AND "Unit1.EmNodes".emFeedback[0].status.initialized AND "Unit1.EmNodes".emFeedback[0].status.homed) OR NOT "Unit1.EmNodes".emFeedback[0].isLinked) AND (("Unit1.EmNodes".emFeedback[1].isLinked AND "Unit1.EmNodes".emFeedback[1].status.initialized AND "Unit1.EmNodes".emFeedback[1].status.homed) OR NOT "Unit1.EmNodes".emFeedback[1].isLinked) AND (("Unit1.EmNodes".emFeedback[2].isLinked AND "Unit1.EmNodes".emFeedback[2].status.initialized AND "Unit1.EmNodes".emFeedback[2].status.homed) OR NOT "Unit1.EmNodes".emFeedback[2].isLinked) AND (("Unit1.EmNodes".emFeedback[3].isLinked AND "Unit1.EmNodes".emFeedback[3].status.initialized AND "Unit1.EmNodes".emFeedback[3].status.homed) OR NOT "Unit1.EmNodes".emFeedback[3].isLinked) AND (("Unit1.EmNodes".emFeedback[4].isLinked AND "Unit1.EmNodes".emFeedback[4].status.initialized AND "Unit1.EmNodes".emFeedback[4].status.homed) OR NOT "Unit1.EmNodes".emFeedback[4].isLinked) AND (("Unit1.EmNodes".emFeedback[5].isLinked AND "Unit1.EmNodes".emFeedback[5].status.initialized AND "Unit1.EmNodes".emFeedback[5].status.homed) OR NOT "Unit1.EmNodes".emFeedback[5].isLinked) AND (("Unit1.EmNodes".emFeedback[6].isLinked AND "Unit1.EmNodes".emFeedback[6].status.initialized AND "Unit1.EmNodes".emFeedback[6].status.homed) OR NOT "Unit1.EmNodes".emFeedback[6].isLinked);
   #statEmHomeScCheck[2] := #_w1 AND (("Unit1.EmNodes".emFeedback[7].isLinked AND "Unit1.EmNodes".emFeedback[7].status.initialized AND "Unit1.EmNodes".emFeedback[7].status.homed) OR NOT "Unit1.EmNodes".emFeedback[7].isLinked) AND (("Unit1.EmNodes".emFeedback[8].isLinked AND "Unit1.EmNodes".emFeedback[8].status.initialized AND "Unit1.EmNodes".emFeedback[8].status.homed) OR NOT "Unit1.EmNodes".emFeedback[8].isLinked) AND (("Unit1.EmNodes".emFeedback[9].isLinked AND "Unit1.EmNodes".emFeedback[9].status.initialized AND "Unit1.EmNodes".emFeedback[9].status.homed) OR NOT "Unit1.EmNodes".emFeedback[9].isLinked) AND (("Unit1.EmNodes".emFeedback[10].isLinked AND "Unit1.EmNodes".emFeedback[10].status.initialized AND "Unit1.EmNodes".emFeedback[10].status.homed) OR NOT "Unit1.EmNodes".emFeedback[10].isLinked) AND (("Unit1.EmNodes".emFeedback[11].isLinked AND "Unit1.EmNodes".emFeedback[11].status.initialized AND "Unit1.EmNodes".emFeedback[11].status.homed) OR NOT "Unit1.EmNodes".emFeedback[11].isLinked) AND (("Unit1.EmNodes".emFeedback[12].isLinked AND "Unit1.EmNodes".emFeedback[12].status.initialized AND "Unit1.EmNodes".emFeedback[12].status.homed) OR NOT "Unit1.EmNodes".emFeedback[12].isLinked) AND (("Unit1.EmNodes".emFeedback[13].isLinked AND "Unit1.EmNodes".emFeedback[13].status.initialized AND "Unit1.EmNodes".emFeedback[13].status.homed) OR NOT "Unit1.EmNodes".emFeedback[13].isLinked);
   #statEmHomeScCheck[0] := #_w1 AND #statEmHomeScCheck[1] AND #statEmHomeScCheck[2];
END_REGION

REGION Network 37: Unit State Commands Execute Enable
   RUNG wire#powerrail
      Contact( #TRUE )
      Contact( #unitInterface.enableControlInterfaces.local )
      Contact( "Unit1.EmNodes".unitStatus.state.starting )
      Contact( #statEmHomeScCheck[0] )
      Contact( "Unit1.ControlNodes".InitializeEnable )
      I_Contact( "Unit1.Alarms".unitAlarms.error )
      Coil( "Unit1.ControlNodes".AutoStartEnable )
      Coil( "Unit1.HmiInterface".AutoStartEnable )
   END_RUNG
   // the same network as SCL:
   "Unit1.ControlNodes".AutoStartEnable := #TRUE AND #unitInterface.enableControlInterfaces.local AND "Unit1.EmNodes".unitStatus.state.starting AND #statEmHomeScCheck[0] AND "Unit1.ControlNodes".InitializeEnable AND NOT "Unit1.Alarms".unitAlarms.error;
   "Unit1.HmiInterface".AutoStartEnable := "Unit1.ControlNodes".AutoStartEnable;
END_REGION

REGION Network 38: Em3 Special Mode End Of Cycle Check
   RUNG wire#powerrail
      Contact( "Unit1.EmNodes".unitStatus.mode.production )
      Contact( "Unit1.EmNodes".unitStatus.state.execute )
      Contact( "Unit1.EmNodes".unitStatus.specialFunctions."End of cycle" )
      wire#w1
      I_Contact( "Unit1.EmNodes".emRelations.em03.cmStatus.TopTapeJRDetect.monitoring.processValue )
      wire#w2
      Coil( #statEOCStatusCheck[3] )
   END_RUNG
   RUNG wire#w1
      Contact( "Unit1.EmNodes".emRelations.em03.sequence.topTapeFixStage.selectJobStatus[5].active )
   END_RUNG wire#w2
   RUNG wire#w1
      Contact( "Unit1.EmNodes".emRelations.em03.sequence.topTapeFixStage.jobInterface.taping1Job3.workingDone )
      Contact( "Unit1.EmNodes".emRelations.em03.sequence.topTapeFixStage.jobInterface.taping2Job4.workingDone )
   END_RUNG wire#w2
   // the same network as SCL:
   #statEOCStatusCheck[3] := "Unit1.EmNodes".unitStatus.mode.production AND "Unit1.EmNodes".unitStatus.state.execute AND "Unit1.EmNodes".unitStatus.specialFunctions."End of cycle" AND (NOT "Unit1.EmNodes".emRelations.em03.cmStatus.TopTapeJRDetect.monitoring.processValue OR "Unit1.EmNodes".emRelations.em03.sequence.topTapeFixStage.selectJobStatus[5].active OR ("Unit1.EmNodes".emRelations.em03.sequence.topTapeFixStage.jobInterface.taping1Job3.workingDone AND "Unit1.EmNodes".emRelations.em03.sequence.topTapeFixStage.jobInterface.taping2Job4.workingDone));
END_REGION

REGION Network 39: Em4 Special Mode End Of Cycle Check
   RUNG wire#powerrail
      Contact( "Unit1.EmNodes".unitStatus.mode.production )
      Contact( "Unit1.EmNodes".unitStatus.state.execute )
      Contact( "Unit1.EmNodes".unitStatus.specialFunctions."End of cycle" )
      wire#w1
      I_Contact( "Unit1.EmNodes".emRelations.em04.cmStatus.SideTapeJRDetect.monitoring.processValue )
      wire#w2
      Coil( #statEOCStatusCheck[4] )
   END_RUNG
   RUNG wire#w1
      Contact( "Unit1.EmNodes".emRelations.em04.sequence.sideTapeFixStage.selectJobStatus[7].active )
   END_RUNG wire#w2
   RUNG wire#w1
      Contact( "Unit1.EmNodes".emRelations.em04.sequence.sideTapeFixStage.jobInterface.taping1Job3.workingDone )
      Contact( "Unit1.EmNodes".emRelations.em04.sequence.sideTapeFixStage.jobInterface.taping2Job4.workingDone )
      Contact( "Unit1.EmNodes".emRelations.em04.sequence.sideTapeFixStage.jobInterface.taping3Job5.workingDone )
      Contact( "Unit1.EmNodes".emRelations.em04.sequence.sideTapeFixStage.jobInterface.taping4Job6.workingDone )
   END_RUNG wire#w2
   // the same network as SCL:
   #statEOCStatusCheck[4] := "Unit1.EmNodes".unitStatus.mode.production AND "Unit1.EmNodes".unitStatus.state.execute AND "Unit1.EmNodes".unitStatus.specialFunctions."End of cycle" AND (NOT "Unit1.EmNodes".emRelations.em04.cmStatus.SideTapeJRDetect.monitoring.processValue OR "Unit1.EmNodes".emRelations.em04.sequence.sideTapeFixStage.selectJobStatus[7].active OR ("Unit1.EmNodes".emRelations.em04.sequence.sideTapeFixStage.jobInterface.taping1Job3.workingDone AND "Unit1.EmNodes".emRelations.em04.sequence.sideTapeFixStage.jobInterface.taping2Job4.workingDone AND "Unit1.EmNodes".emRelations.em04.sequence.sideTapeFixStage.jobInterface.taping3Job5.workingDone AND "Unit1.EmNodes".emRelations.em04.sequence.sideTapeFixStage.jobInterface.taping4Job6.workingDone));
END_REGION

REGION Network 40: Em6 Special Mode End Of Cycle Check
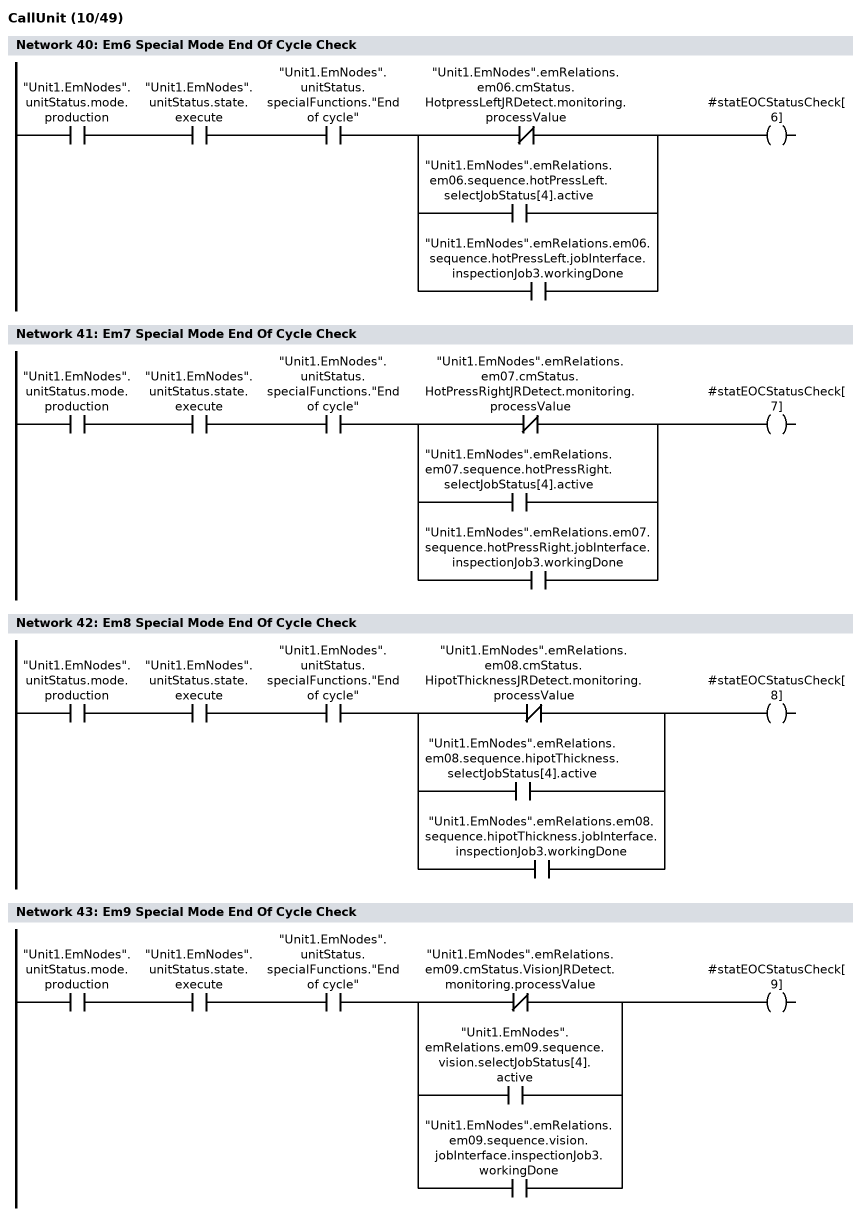
   RUNG wire#powerrail
      Contact( "Unit1.EmNodes".unitStatus.mode.production )
      Contact( "Unit1.EmNodes".unitStatus.state.execute )
      Contact( "Unit1.EmNodes".unitStatus.specialFunctions."End of cycle" )
      wire#w1
      I_Contact( "Unit1.EmNodes".emRelations.em06.cmStatus.HotpressLeftJRDetect.monitoring.processValue )
      wire#w2
      Coil( #statEOCStatusCheck[6] )
   END_RUNG
   RUNG wire#w1
      Contact( "Unit1.EmNodes".emRelations.em06.sequence.hotPressLeft.selectJobStatus[4].active )
   END_RUNG wire#w2
   RUNG wire#w1
      Contact( "Unit1.EmNodes".emRelations.em06.sequence.hotPressLeft.jobInterface.inspectionJob3.workingDone )
   END_RUNG wire#w2
   // the same network as SCL:
   #statEOCStatusCheck[6] := "Unit1.EmNodes".unitStatus.mode.production AND "Unit1.EmNodes".unitStatus.state.execute AND "Unit1.EmNodes".unitStatus.specialFunctions."End of cycle" AND (NOT "Unit1.EmNodes".emRelations.em06.cmStatus.HotpressLeftJRDetect.monitoring.processValue OR "Unit1.EmNodes".emRelations.em06.sequence.hotPressLeft.selectJobStatus[4].active OR "Unit1.EmNodes".emRelations.em06.sequence.hotPressLeft.jobInterface.inspectionJob3.workingDone);
END_REGION

REGION Network 41: Em7 Special Mode End Of Cycle Check
   RUNG wire#powerrail
      Contact( "Unit1.EmNodes".unitStatus.mode.production )
      Contact( "Unit1.EmNodes".unitStatus.state.execute )
      Contact( "Unit1.EmNodes".unitStatus.specialFunctions."End of cycle" )
      wire#w1
      I_Contact( "Unit1.EmNodes".emRelations.em07.cmStatus.HotPressRightJRDetect.monitoring.processValue )
      wire#w2
      Coil( #statEOCStatusCheck[7] )
   END_RUNG
   RUNG wire#w1
      Contact( "Unit1.EmNodes".emRelations.em07.sequence.hotPressRight.selectJobStatus[4].active )
   END_RUNG wire#w2
   RUNG wire#w1
      Contact( "Unit1.EmNodes".emRelations.em07.sequence.hotPressRight.jobInterface.inspectionJob3.workingDone )
   END_RUNG wire#w2
   // the same network as SCL:
   #statEOCStatusCheck[7] := "Unit1.EmNodes".unitStatus.mode.production AND "Unit1.EmNodes".unitStatus.state.execute AND "Unit1.EmNodes".unitStatus.specialFunctions."End of cycle" AND (NOT "Unit1.EmNodes".emRelations.em07.cmStatus.HotPressRightJRDetect.monitoring.processValue OR "Unit1.EmNodes".emRelations.em07.sequence.hotPressRight.selectJobStatus[4].active OR "Unit1.EmNodes".emRelations.em07.sequence.hotPressRight.jobInterface.inspectionJob3.workingDone);
END_REGION

REGION Network 42: Em8 Special Mode End Of Cycle Check
   RUNG wire#powerrail
      Contact( "Unit1.EmNodes".unitStatus.mode.production )
      Contact( "Unit1.EmNodes".unitStatus.state.execute )
      Contact( "Unit1.EmNodes".unitStatus.specialFunctions."End of cycle" )
      wire#w1
      I_Contact( "Unit1.EmNodes".emRelations.em08.cmStatus.HipotThicknessJRDetect.monitoring.processValue )
      wire#w2
      Coil( #statEOCStatusCheck[8] )
   END_RUNG
   RUNG wire#w1
      Contact( "Unit1.EmNodes".emRelations.em08.sequence.hipotThickness.selectJobStatus[4].active )
   END_RUNG wire#w2
   RUNG wire#w1
      Contact( "Unit1.EmNodes".emRelations.em08.sequence.hipotThickness.jobInterface.inspectionJob3.workingDone )
   END_RUNG wire#w2
   // the same network as SCL:
   #statEOCStatusCheck[8] := "Unit1.EmNodes".unitStatus.mode.production AND "Unit1.EmNodes".unitStatus.state.execute AND "Unit1.EmNodes".unitStatus.specialFunctions."End of cycle" AND (NOT "Unit1.EmNodes".emRelations.em08.cmStatus.HipotThicknessJRDetect.monitoring.processValue OR "Unit1.EmNodes".emRelations.em08.sequence.hipotThickness.selectJobStatus[4].active OR "Unit1.EmNodes".emRelations.em08.sequence.hipotThickness.jobInterface.inspectionJob3.workingDone);
END_REGION

REGION Network 43: Em9 Special Mode End Of Cycle Check
   RUNG wire#powerrail
      Contact( "Unit1.EmNodes".unitStatus.mode.production )
      Contact( "Unit1.EmNodes".unitStatus.state.execute )
      Contact( "Unit1.EmNodes".unitStatus.specialFunctions."End of cycle" )
      wire#w1
      I_Contact( "Unit1.EmNodes".emRelations.em09.cmStatus.VisionJRDetect.monitoring.processValue )
      wire#w2
      Coil( #statEOCStatusCheck[9] )
   END_RUNG
   RUNG wire#w1
      Contact( "Unit1.EmNodes".emRelations.em09.sequence.vision.selectJobStatus[4].active )
   END_RUNG wire#w2
   RUNG wire#w1
      Contact( "Unit1.EmNodes".emRelations.em09.sequence.vision.jobInterface.inspectionJob3.workingDone )
   END_RUNG wire#w2
   // the same network as SCL:
   #statEOCStatusCheck[9] := "Unit1.EmNodes".unitStatus.mode.production AND "Unit1.EmNodes".unitStatus.state.execute AND "Unit1.EmNodes".unitStatus.specialFunctions."End of cycle" AND (NOT "Unit1.EmNodes".emRelations.em09.cmStatus.VisionJRDetect.monitoring.processValue OR "Unit1.EmNodes".emRelations.em09.sequence.vision.selectJobStatus[4].active OR "Unit1.EmNodes".emRelations.em09.sequence.vision.jobInterface.inspectionJob3.workingDone);
END_REGION

REGION Network 44: Em10 Special Mode End Of Cycle Check
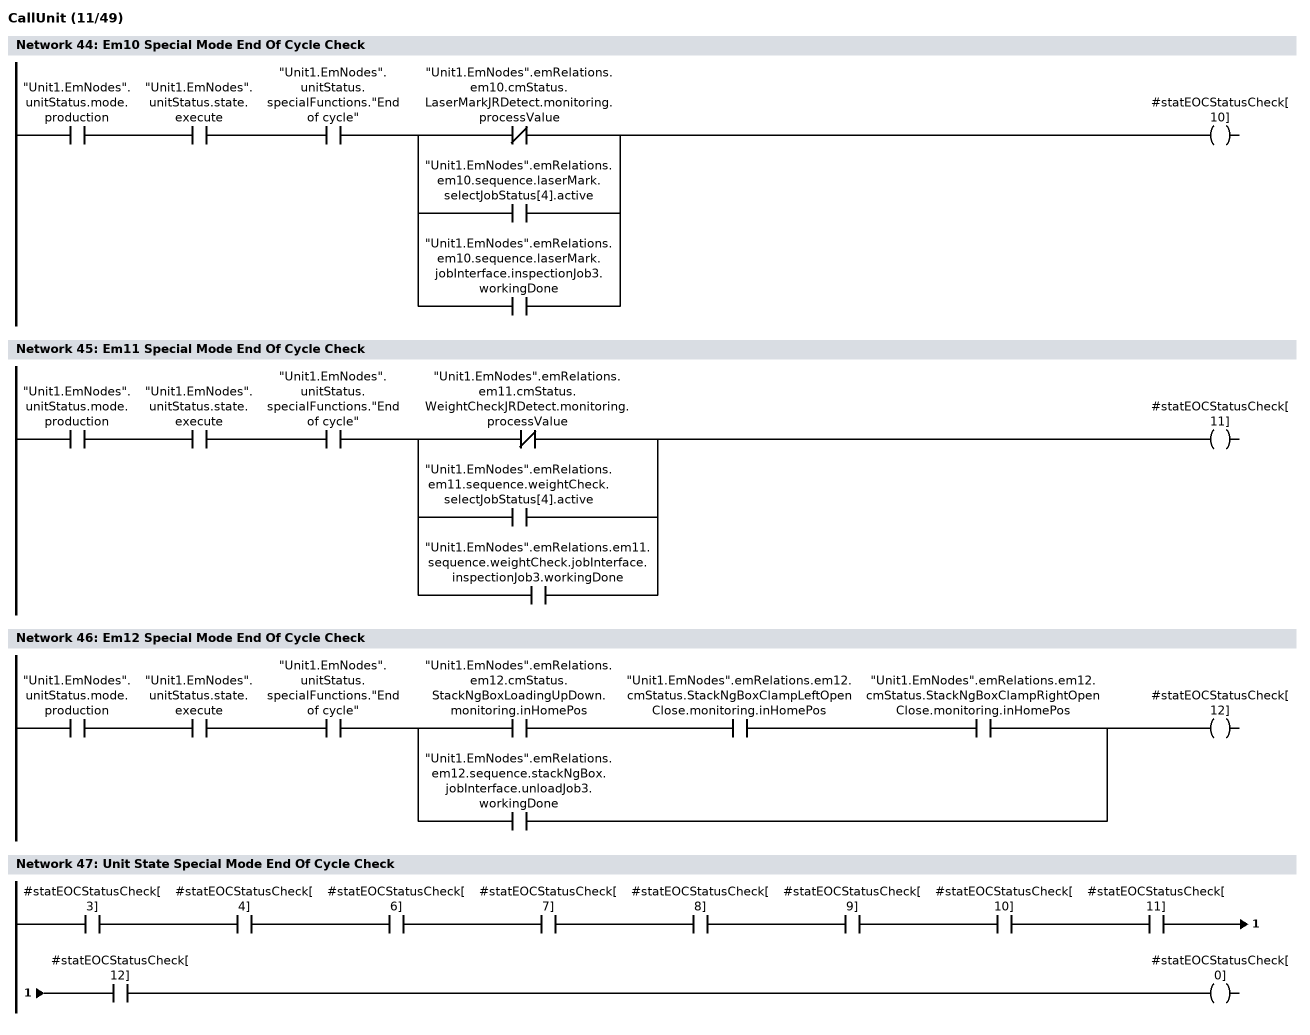
   RUNG wire#powerrail
      Contact( "Unit1.EmNodes".unitStatus.mode.production )
      Contact( "Unit1.EmNodes".unitStatus.state.execute )
      Contact( "Unit1.EmNodes".unitStatus.specialFunctions."End of cycle" )
      wire#w1
      I_Contact( "Unit1.EmNodes".emRelations.em10.cmStatus.LaserMarkJRDetect.monitoring.processValue )
      wire#w2
      Coil( #statEOCStatusCheck[10] )
   END_RUNG
   RUNG wire#w1
      Contact( "Unit1.EmNodes".emRelations.em10.sequence.laserMark.selectJobStatus[4].active )
   END_RUNG wire#w2
   RUNG wire#w1
      Contact( "Unit1.EmNodes".emRelations.em10.sequence.laserMark.jobInterface.inspectionJob3.workingDone )
   END_RUNG wire#w2
   // the same network as SCL:
   #statEOCStatusCheck[10] := "Unit1.EmNodes".unitStatus.mode.production AND "Unit1.EmNodes".unitStatus.state.execute AND "Unit1.EmNodes".unitStatus.specialFunctions."End of cycle" AND (NOT "Unit1.EmNodes".emRelations.em10.cmStatus.LaserMarkJRDetect.monitoring.processValue OR "Unit1.EmNodes".emRelations.em10.sequence.laserMark.selectJobStatus[4].active OR "Unit1.EmNodes".emRelations.em10.sequence.laserMark.jobInterface.inspectionJob3.workingDone);
END_REGION

REGION Network 45: Em11 Special Mode End Of Cycle Check
   RUNG wire#powerrail
      Contact( "Unit1.EmNodes".unitStatus.mode.production )
      Contact( "Unit1.EmNodes".unitStatus.state.execute )
      Contact( "Unit1.EmNodes".unitStatus.specialFunctions."End of cycle" )
      wire#w1
      I_Contact( "Unit1.EmNodes".emRelations.em11.cmStatus.WeightCheckJRDetect.monitoring.processValue )
      wire#w2
      Coil( #statEOCStatusCheck[11] )
   END_RUNG
   RUNG wire#w1
      Contact( "Unit1.EmNodes".emRelations.em11.sequence.weightCheck.selectJobStatus[4].active )
   END_RUNG wire#w2
   RUNG wire#w1
      Contact( "Unit1.EmNodes".emRelations.em11.sequence.weightCheck.jobInterface.inspectionJob3.workingDone )
   END_RUNG wire#w2
   // the same network as SCL:
   #statEOCStatusCheck[11] := "Unit1.EmNodes".unitStatus.mode.production AND "Unit1.EmNodes".unitStatus.state.execute AND "Unit1.EmNodes".unitStatus.specialFunctions."End of cycle" AND (NOT "Unit1.EmNodes".emRelations.em11.cmStatus.WeightCheckJRDetect.monitoring.processValue OR "Unit1.EmNodes".emRelations.em11.sequence.weightCheck.selectJobStatus[4].active OR "Unit1.EmNodes".emRelations.em11.sequence.weightCheck.jobInterface.inspectionJob3.workingDone);
END_REGION

REGION Network 46: Em12 Special Mode End Of Cycle Check
   RUNG wire#powerrail
      Contact( "Unit1.EmNodes".unitStatus.mode.production )
      Contact( "Unit1.EmNodes".unitStatus.state.execute )
      Contact( "Unit1.EmNodes".unitStatus.specialFunctions."End of cycle" )
      wire#w1
      Contact( "Unit1.EmNodes".emRelations.em12.cmStatus.StackNgBoxLoadingUpDown.monitoring.inHomePos )
      Contact( "Unit1.EmNodes".emRelations.em12.cmStatus.StackNgBoxClampLeftOpenClose.monitoring.inHomePos )
      Contact( "Unit1.EmNodes".emRelations.em12.cmStatus.StackNgBoxClampRightOpenClose.monitoring.inHomePos )
      wire#w2
      Coil( #statEOCStatusCheck[12] )
   END_RUNG
   RUNG wire#w1
      Contact( "Unit1.EmNodes".emRelations.em12.sequence.stackNgBox.jobInterface.unloadJob3.workingDone )
   END_RUNG wire#w2
   // the same network as SCL:
   #statEOCStatusCheck[12] := "Unit1.EmNodes".unitStatus.mode.production AND "Unit1.EmNodes".unitStatus.state.execute AND "Unit1.EmNodes".unitStatus.specialFunctions."End of cycle" AND (("Unit1.EmNodes".emRelations.em12.cmStatus.StackNgBoxLoadingUpDown.monitoring.inHomePos AND "Unit1.EmNodes".emRelations.em12.cmStatus.StackNgBoxClampLeftOpenClose.monitoring.inHomePos AND "Unit1.EmNodes".emRelations.em12.cmStatus.StackNgBoxClampRightOpenClose.monitoring.inHomePos) OR "Unit1.EmNodes".emRelations.em12.sequence.stackNgBox.jobInterface.unloadJob3.workingDone);
END_REGION

REGION Network 47: Unit State Special Mode End Of Cycle Check
   RUNG wire#powerrail
      Contact( #statEOCStatusCheck[3] )
      Contact( #statEOCStatusCheck[4] )
      Contact( #statEOCStatusCheck[6] )
      Contact( #statEOCStatusCheck[7] )
      Contact( #statEOCStatusCheck[8] )
      Contact( #statEOCStatusCheck[9] )
      Contact( #statEOCStatusCheck[10] )
      Contact( #statEOCStatusCheck[11] )
      Contact( #statEOCStatusCheck[12] )
      Coil( #statEOCStatusCheck[0] )
   END_RUNG
   // the same network as SCL:
   #statEOCStatusCheck[0] := #statEOCStatusCheck[3] AND #statEOCStatusCheck[4] AND #statEOCStatusCheck[6] AND #statEOCStatusCheck[7] AND #statEOCStatusCheck[8] AND #statEOCStatusCheck[9] AND #statEOCStatusCheck[10] AND #statEOCStatusCheck[11] AND #statEOCStatusCheck[12];
END_REGION

REGION Network 48: Unit State Special Mode Run Out Check
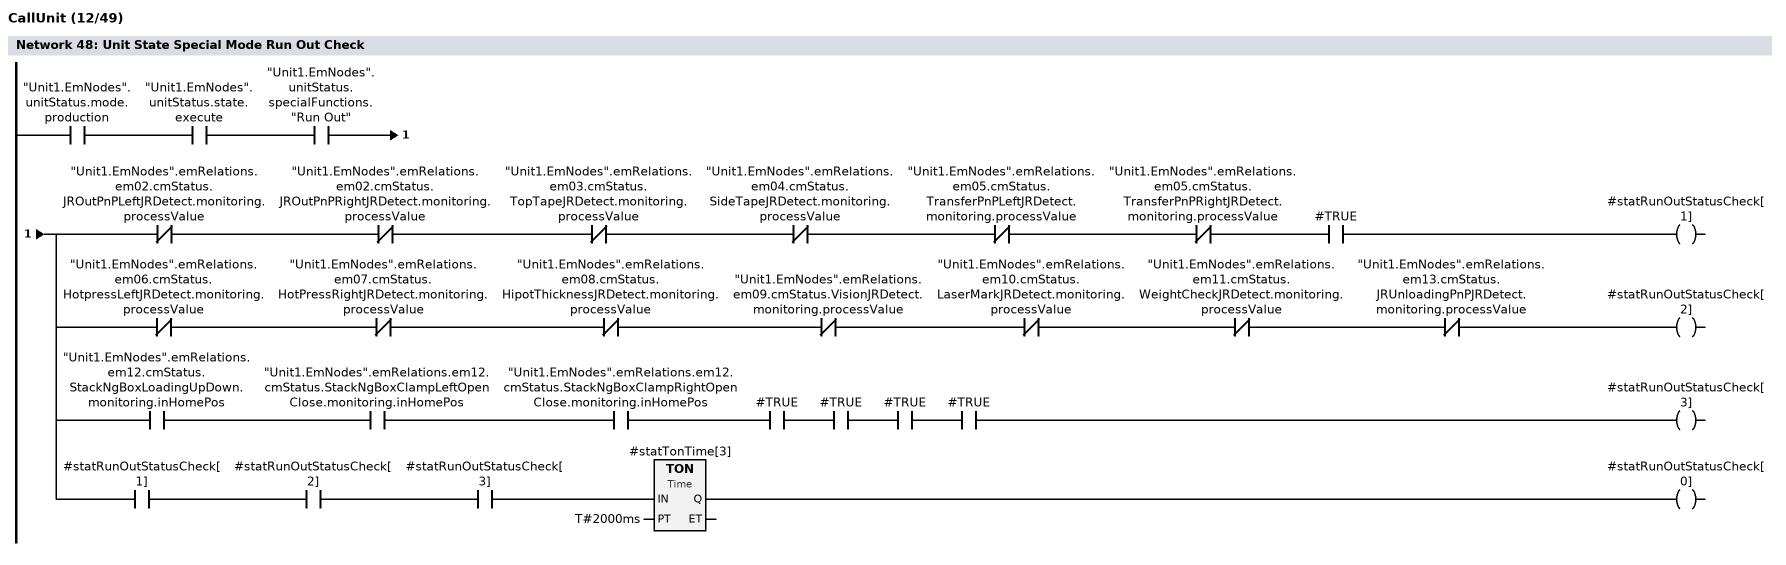
   RUNG wire#powerrail
      Contact( "Unit1.EmNodes".unitStatus.mode.production )
      Contact( "Unit1.EmNodes".unitStatus.state.execute )
      Contact( "Unit1.EmNodes".unitStatus.specialFunctions."Run Out" )
      wire#w1
      I_Contact( "Unit1.EmNodes".emRelations.em02.cmStatus.JROutPnPLeftJRDetect.monitoring.processValue )
      I_Contact( "Unit1.EmNodes".emRelations.em02.cmStatus.JROutPnPRightJRDetect.monitoring.processValue )
      I_Contact( "Unit1.EmNodes".emRelations.em03.cmStatus.TopTapeJRDetect.monitoring.processValue )
      I_Contact( "Unit1.EmNodes".emRelations.em04.cmStatus.SideTapeJRDetect.monitoring.processValue )
      I_Contact( "Unit1.EmNodes".emRelations.em05.cmStatus.TransferPnPLeftJRDetect.monitoring.processValue )
      I_Contact( "Unit1.EmNodes".emRelations.em05.cmStatus.TransferPnPRightJRDetect.monitoring.processValue )
      Contact( #TRUE )
      Coil( #statRunOutStatusCheck[1] )
   END_RUNG
   RUNG wire#w1
      I_Contact( "Unit1.EmNodes".emRelations.em06.cmStatus.HotpressLeftJRDetect.monitoring.processValue )
      I_Contact( "Unit1.EmNodes".emRelations.em07.cmStatus.HotPressRightJRDetect.monitoring.processValue )
      I_Contact( "Unit1.EmNodes".emRelations.em08.cmStatus.HipotThicknessJRDetect.monitoring.processValue )
      I_Contact( "Unit1.EmNodes".emRelations.em09.cmStatus.VisionJRDetect.monitoring.processValue )
      I_Contact( "Unit1.EmNodes".emRelations.em10.cmStatus.LaserMarkJRDetect.monitoring.processValue )
      I_Contact( "Unit1.EmNodes".emRelations.em11.cmStatus.WeightCheckJRDetect.monitoring.processValue )
      I_Contact( "Unit1.EmNodes".emRelations.em13.cmStatus.JRUnloadingPnPJRDetect.monitoring.processValue )
      Coil( #statRunOutStatusCheck[2] )
   END_RUNG
   RUNG wire#w1
      Contact( "Unit1.EmNodes".emRelations.em12.cmStatus.StackNgBoxLoadingUpDown.monitoring.inHomePos )
      Contact( "Unit1.EmNodes".emRelations.em12.cmStatus.StackNgBoxClampLeftOpenClose.monitoring.inHomePos )
      Contact( "Unit1.EmNodes".emRelations.em12.cmStatus.StackNgBoxClampRightOpenClose.monitoring.inHomePos )
      Contact( #TRUE )
      Contact( #TRUE )
      Contact( #TRUE )
      Contact( #TRUE )
      Coil( #statRunOutStatusCheck[3] )
   END_RUNG
   RUNG wire#w1
      Contact( #statRunOutStatusCheck[1] )
      Contact( #statRunOutStatusCheck[2] )
      Contact( #statRunOutStatusCheck[3] )
      { S7_Templates := "time_type := Time" } #statTonTime[3].TON(pt := T#2000ms, et =>)
      Coil( #statRunOutStatusCheck[0] )
   END_RUNG
   // the same network as SCL:
   #_w1 := "Unit1.EmNodes".unitStatus.mode.production AND "Unit1.EmNodes".unitStatus.state.execute AND "Unit1.EmNodes".unitStatus.specialFunctions."Run Out";
   #statRunOutStatusCheck[1] := #_w1 AND NOT "Unit1.EmNodes".emRelations.em02.cmStatus.JROutPnPLeftJRDetect.monitoring.processValue AND NOT "Unit1.EmNodes".emRelations.em02.cmStatus.JROutPnPRightJRDetect.monitoring.processValue AND NOT "Unit1.EmNodes".emRelations.em03.cmStatus.TopTapeJRDetect.monitoring.processValue AND NOT "Unit1.EmNodes".emRelations.em04.cmStatus.SideTapeJRDetect.monitoring.processValue AND NOT "Unit1.EmNodes".emRelations.em05.cmStatus.TransferPnPLeftJRDetect.monitoring.processValue AND NOT "Unit1.EmNodes".emRelations.em05.cmStatus.TransferPnPRightJRDetect.monitoring.processValue AND #TRUE;
   #statRunOutStatusCheck[2] := #_w1 AND NOT "Unit1.EmNodes".emRelations.em06.cmStatus.HotpressLeftJRDetect.monitoring.processValue AND NOT "Unit1.EmNodes".emRelations.em07.cmStatus.HotPressRightJRDetect.monitoring.processValue AND NOT "Unit1.EmNodes".emRelations.em08.cmStatus.HipotThicknessJRDetect.monitoring.processValue AND NOT "Unit1.EmNodes".emRelations.em09.cmStatus.VisionJRDetect.monitoring.processValue AND NOT "Unit1.EmNodes".emRelations.em10.cmStatus.LaserMarkJRDetect.monitoring.processValue AND NOT "Unit1.EmNodes".emRelations.em11.cmStatus.WeightCheckJRDetect.monitoring.processValue AND NOT "Unit1.EmNodes".emRelations.em13.cmStatus.JRUnloadingPnPJRDetect.monitoring.processValue;
   #statRunOutStatusCheck[3] := #_w1 AND "Unit1.EmNodes".emRelations.em12.cmStatus.StackNgBoxLoadingUpDown.monitoring.inHomePos AND "Unit1.EmNodes".emRelations.em12.cmStatus.StackNgBoxClampLeftOpenClose.monitoring.inHomePos AND "Unit1.EmNodes".emRelations.em12.cmStatus.StackNgBoxClampRightOpenClose.monitoring.inHomePos AND #TRUE AND #TRUE AND #TRUE AND #TRUE;
   #statTonTime[3].TON(IN := #_w1 AND #statRunOutStatusCheck[1] AND #statRunOutStatusCheck[2] AND #statRunOutStatusCheck[3],
                       PT := T#2000ms);
   #statRunOutStatusCheck[0] := #statTonTime[3].Q;
END_REGION

